METHOD PUBLIC Clone : I_Node
VAR
    pNode : POINTER TO Node_F_VN_ConvertMaps;
END_VAR
pNode := __NEW(Node_F_VN_ConvertMaps);
Clone := pNode^;
END_METHOD

METHOD PROTECTED OnExecute
hresult.Value := F_VN_ConvertMaps(
    ipSrcMap1 := ipSrcMap1.Value,
    ipSrcMap2 := ipSrcMap2.Value,
    ipDestMap1 := ipDestMap1.Value,
    ipDestMap2 := ipDestMap2.Value,
    eDestMap1Type := eDestMap1Type.Value,
    nDestMap1Channels := nDestMap1Channels.Value,
    hrPrev := hrPrev.Value);
END_METHOD

METHOD PUBLIC PreExecutionCheck
VAR_INPUT
    Check : I_PreExecutionChecks;
END_VAR
Check.IsTrue(IsRemapMapPairValid(ipSrcMap1.Value, ipSrcMap2.Value), 'Unsupported source map pair: use REAL XY, separate REAL X/Y, or INT XY with optional UINT coefficients');
Check.IsTrue((eDestMap1Type.Value = ETcVnElementType.TCVN_ET_REAL) OR
             (eDestMap1Type.Value = ETcVnElementType.TCVN_ET_INT), 'Destination map type must be REAL or INT');
Check.IsTrue((nDestMap1Channels.Value = 1) OR (nDestMap1Channels.Value = 2), 'Destination map must have 1 or 2 channels');
Check.IsTrue((eDestMap1Type.Value <> ETcVnElementType.TCVN_ET_INT) OR
             (nDestMap1Channels.Value = 2), 'Fixed-point destination map must have 2 channels');
Check.IsTrue((ipDestMap1.Value = 0) OR ((ipDestMap1.Value <> ipSrcMap1.Value) AND (ipDestMap1.Value <> ipSrcMap2.Value)), 'ipDestMap1 must be different from the source maps');
Check.IsTrue((ipDestMap2.Value = 0) OR ((ipDestMap2.Value <> ipSrcMap1.Value) AND (ipDestMap2.Value <> ipSrcMap2.Value)), 'ipDestMap2 must be different from the source maps');
Check.IsTrue((ipDestMap1.Value = 0) OR (ipDestMap1.Value <> ipDestMap2.Value), 'Destination maps must be different images');
END_METHOD

END_FUNCTION_BLOCK

// Nodes/Geometric and Coord Transform/Node_F_VN_ConvertPolarToCartesianImages
{attribute 'linkalways'}
{attribute 'no_explicit_call' := 'This FB is a CLASS and must be accessed using methods or properties'}
{attribute 'enable_dynamic_creation'}
FUNCTION_BLOCK Node_F_VN_ConvertPolarToCartesianImages EXTENDS VisionNode
VAR
    ipSrcImageMag : _ITcVnImage;
    ipSrcImageAng : _ITcVnImage;
    ipDestImageX : _ITcVnImage;
    ipDestImageY : _ITcVnImage;
    hrPrev : _HRESULT(S_OK);
    hresult : _HRESULT(S_OK);
END_VAR

METHOD FB_init : BOOL
VAR_INPUT
    bInitRetains : BOOL;
    bInCopyCode : BOOL;
END_VAR
AddInput('ipSrcImageMag', ipSrcImageMag);
AddInput('ipSrcImageAng', ipSrcImageAng);
AddOutput('ipDestImageX', ipDestImageX);
AddOutput('ipDestImageY', ipDestImageY);
AddInput('hrPrev', hrPrev);
AddOutput('hresult', hresult);
END_METHOD

METHOD PUBLIC Clone : I_Node
VAR
    pNode : POINTER TO Node_F_VN_ConvertPolarToCartesianImages;
END_VAR
pNode := __NEW(Node_F_VN_ConvertPolarToCartesianImages);
Clone := pNode^;
END_METHOD

METHOD PROTECTED OnExecute
hresult.Value := F_VN_ConvertPolarToCartesianImages(
    ipSrcImageMag := ipSrcImageMag.Value,
    ipSrcImageAng := ipSrcImageAng.Value,
    ipDestImageX := ipDestImageX.Value,
    ipDestImageY := ipDestImageY.Value,
    hrPrev := hrPrev.Value);
END_METHOD

METHOD PUBLIC PreExecutionCheck
VAR_INPUT
    Check : I_PreExecutionChecks;
END_VAR
Check.IsTrue(ipSrcImageMag.IsValid, 'ipSrcImageMag must contain an image');
Check.IsTrue(ipSrcImageMag.IsElementType(ETcVnElementType.TCVN_ET_REAL) OR
             ipSrcImageMag.IsElementType(ETcVnElementType.TCVN_ET_LREAL), 'Coordinate images must contain REAL or LREAL elements');
Check.IsTrue(ipSrcImageAng.IsValid, 'ipSrcImageAng must contain an image');
Check.IsTrue(ImagesHaveMatchingPixelFormats(ipSrcImageMag.Value, ipSrcImageAng.Value), 'Source images must have matching pixel formats');
Check.IsTrue(IsImage1SizeEqualToImage2Size(ipSrcImageMag.Value, ipSrcImageAng.Value), 'Source images must have matching dimensions');
END_METHOD

END_FUNCTION_BLOCK

// Nodes/Geometric and Coord Transform/Node_F_VN_ConvertPolarToCartesianImagesExp
{attribute 'linkalways'}
{attribute 'no_explicit_call' := 'This FB is a CLASS and must be accessed using methods or properties'}
{attribute 'enable_dynamic_creation'}
FUNCTION_BLOCK Node_F_VN_ConvertPolarToCartesianImagesExp EXTENDS VisionNode
VAR
    ipSrcImageMag : _ITcVnImage;
    ipSrcImageAng : _ITcVnImage;
    ipDestImageX : _ITcVnImage;
    ipDestImageY : _ITcVnImage;
    bAngleInDegrees : _BOOL(FALSE);
    hrPrev : _HRESULT(S_OK);
    hresult : _HRESULT(S_OK);
END_VAR

METHOD FB_init : BOOL
VAR_INPUT
    bInitRetains : BOOL;
    bInCopyCode : BOOL;
END_VAR
AddInput('ipSrcImageMag', ipSrcImageMag);
AddInput('ipSrcImageAng', ipSrcImageAng);
AddOutput('ipDestImageX', ipDestImageX);
AddOutput('ipDestImageY', ipDestImageY);
AddParameter('bAngleInDegrees', bAngleInDegrees);
AddInput('hrPrev', hrPrev);
AddOutput('hresult', hresult);
END_METHOD

METHOD PUBLIC Clone : I_Node
VAR
    pNode : POINTER TO Node_F_VN_ConvertPolarToCartesianImagesExp;
END_VAR
pNode := __NEW(Node_F_VN_ConvertPolarToCartesianImagesExp);
Clone := pNode^;
END_METHOD

METHOD PROTECTED OnExecute
hresult.Value := F_VN_ConvertPolarToCartesianImagesExp(
    ipSrcImageMag := ipSrcImageMag.Value,
    ipSrcImageAng := ipSrcImageAng.Value,
    ipDestImageX := ipDestImageX.Value,
    ipDestImageY := ipDestImageY.Value,
    bAngleInDegrees := bAngleInDegrees.Value,
    hrPrev := hrPrev.Value);
END_METHOD

METHOD PUBLIC PreExecutionCheck
VAR_INPUT
    Check : I_PreExecutionChecks;
END_VAR
Check.IsTrue(ipSrcImageMag.IsValid, 'ipSrcImageMag must contain an image');
Check.IsTrue(ipSrcImageMag.IsElementType(ETcVnElementType.TCVN_ET_REAL) OR
             ipSrcImageMag.IsElementType(ETcVnElementType.TCVN_ET_LREAL), 'Coordinate images must contain REAL or LREAL elements');
Check.IsTrue(ipSrcImageAng.IsValid, 'ipSrcImageAng must contain an image');
Check.IsTrue(ImagesHaveMatchingPixelFormats(ipSrcImageMag.Value, ipSrcImageAng.Value), 'Source images must have matching pixel formats');
Check.IsTrue(IsImage1SizeEqualToImage2Size(ipSrcImageMag.Value, ipSrcImageAng.Value), 'Source images must have matching dimensions');
END_METHOD

END_FUNCTION_BLOCK

// Nodes/Geometric and Coord Transform/Node_F_VN_ConvertPolarToCartesianPoints
{attribute 'linkalways'} 
{attribute 'no_explicit_call' := 'This FB is a CLASS and must be accessed using methods or properties'}
{attribute 'enable_dynamic_creation'}
FUNCTION_BLOCK Node_F_VN_ConvertPolarToCartesianPoints EXTENDS VisionNode
VAR
	ipSrcPointsPolar : _ITcVnContainer;
    ipDestPointsCart : _ITcVnContainer;
    hrPrev : _HRESULT(S_OK);
	hresult : _HRESULT(S_OK);
END_VAR

METHOD FB_init : BOOL
VAR_INPUT
	bInitRetains : BOOL; // if TRUE, the retain variables are initialized (warm start / cold start)
	bInCopyCode : BOOL;  // if TRUE, the instance afterwards gets moved into the copy code (online change)
END_VAR
AddInput('ipSrcPointsPolar', ipSrcPointsPolar);
AddInput('hrPrev', hrPrev);
AddOutput('ipDestPointsCart', ipDestPointsCart);
AddOutput('hresult',hresult);
END_METHOD

METHOD PUBLIC  Clone : I_Node
VAR
	pNode : POINTER TO Node_F_VN_ConvertPolarToCartesianPoints;
END_VAR
pNode := __NEW(Node_F_VN_ConvertPolarToCartesianPoints);
Clone := pNode^;
END_METHOD

METHOD PROTECTED OnExecute
hresult.Value := F_VN_ConvertPolarToCartesianPoints(
	ipSrcPointsPolar := ipSrcPointsPolar.Value,
	ipDestPointsCart := ipDestPointsCart.Value,
	hrPrev := hrPrev.Value);
END_METHOD

METHOD PUBLIC PreExecutionCheck
VAR_INPUT
	Check : I_PreExecutionChecks;
END_VAR
Check.IsTrue(ipSrcPointsPolar.IsValid, 'ipSrcPointsPolar must be a valid container');
Check.IsTrue((ipSrcPointsPolar.IsType(TC_GLOBAL_CONST_LIST.ContainerType_Vector_TcVnPoint2_REAL) OR
              ipSrcPointsPolar.IsType(TC_GLOBAL_CONST_LIST.ContainerType_Vector_TcVnPoint2_LREAL)),
              'ipSrcPointsPolar contains incorrect type');
END_METHOD

END_FUNCTION_BLOCK

// Nodes/Geometric and Coord Transform/Node_F_VN_ConvertPolarToCartesianPointsExp
{attribute 'linkalways'} 
{attribute 'no_explicit_call' := 'This FB is a CLASS and must be accessed using methods or properties'}
{attribute 'enable_dynamic_creation'}
FUNCTION_BLOCK Node_F_VN_ConvertPolarToCartesianPointsExp EXTENDS VisionNode
VAR
	ipSrcPointsPolar : _ITcVnContainer;
    ipDestPointsCart : _ITcVnContainer;
    bAngleInDegrees : _BOOL(FALSE);
    hrPrev : _HRESULT(S_OK);
	hresult : _HRESULT(S_OK);
END_VAR

METHOD FB_init : BOOL
VAR_INPUT
	bInitRetains : BOOL; // if TRUE, the retain variables are initialized (warm start / cold start)
	bInCopyCode : BOOL;  // if TRUE, the instance afterwards gets moved into the copy code (online change)
END_VAR
AddInput('ipSrcPointsPolar', ipSrcPointsPolar);
AddParameter('bAngleInDegrees', bAngleInDegrees);
AddInput('hrPrev', hrPrev);
AddOutput('ipDestPointsCart', ipDestPointsCart);
AddOutput('hresult',hresult);
END_METHOD

METHOD PUBLIC  Clone : I_Node
VAR
	pNode : POINTER TO Node_F_VN_ConvertPolarToCartesianPointsExp;
END_VAR
pNode := __NEW(Node_F_VN_ConvertPolarToCartesianPointsExp);
Clone := pNode^;
END_METHOD

METHOD PROTECTED OnExecute
hresult.Value := F_VN_ConvertPolarToCartesianPointsExp(
	ipSrcPointsPolar := ipSrcPointsPolar.Value,
	ipDestPointsCart := ipDestPointsCart.Value,
    bAngleInDegrees := bAngleInDegrees.Value,
	hrPrev := hrPrev.Value);
END_METHOD

METHOD PUBLIC PreExecutionCheck
VAR_INPUT
	Check : I_PreExecutionChecks;
END_VAR
Check.IsTrue(ipSrcPointsPolar.IsValid, 'ipSrcPointsPolar must be a valid container');
Check.IsTrue((ipSrcPointsPolar.IsType(TC_GLOBAL_CONST_LIST.ContainerType_Vector_TcVnPoint2_REAL) OR
              ipSrcPointsPolar.IsType(TC_GLOBAL_CONST_LIST.ContainerType_Vector_TcVnPoint2_LREAL)),
              'ipSrcPointsPolar contains incorrect type');
END_METHOD

END_FUNCTION_BLOCK

// Nodes/Geometric and Coord Transform/Node_F_VN_DecomposeAffineTransformation
{attribute 'linkalways'} 
{attribute 'no_explicit_call' := 'This FB is a CLASS and must be accessed using methods or properties'}
{attribute 'enable_dynamic_creation'}
FUNCTION_BLOCK Node_F_VN_DecomposeAffineTransformation EXTENDS VisionNode
VAR
    aAffineTransform : _TcVnMatrix2x3_LREAL;
    fRotationAngle : _LREAL(0.0);
    hrPrev : _HRESULT(S_OK);
	hresult : _HRESULT(S_OK);
END_VAR

METHOD FB_init : BOOL
VAR_INPUT
	bInitRetains : BOOL; // if TRUE, the retain variables are initialized (warm start / cold start)
	bInCopyCode : BOOL;  // if TRUE, the instance afterwards gets moved into the copy code (online change)
END_VAR
AddInput('aAffineTransform', aAffineTransform);
AddInput('hrPrev', hrPrev);
AddOutput('fRotationAngle', fRotationAngle);
AddOutput('hresult',hresult);
END_METHOD

METHOD PUBLIC  Clone : I_Node
VAR
	pNode : POINTER TO Node_F_VN_DecomposeAffineTransformation;
END_VAR
pNode := __NEW(Node_F_VN_DecomposeAffineTransformation);
Clone := pNode^;
END_METHOD

METHOD PROTECTED OnExecute
hresult.Value := F_VN_DecomposeAffineTransformation(
	aAffineTransform := aAffineTransform.Value, 
	fRotationAngle := fRotationAngle.Value, 
	hrPrev := hrPrev.Value);
END_METHOD

METHOD PUBLIC PreExecutionCheck
VAR_INPUT
	Check : I_PreExecutionChecks;
END_VAR
END_METHOD

END_FUNCTION_BLOCK

// Nodes/Geometric and Coord Transform/Node_F_VN_DecomposeAffineTransformationExp
{attribute 'linkalways'} 
{attribute 'no_explicit_call' := 'This FB is a CLASS and must be accessed using methods or properties'}
{attribute 'enable_dynamic_creation'}
FUNCTION_BLOCK Node_F_VN_DecomposeAffineTransformationExp EXTENDS VisionNode
VAR
    aAffineTransform : _TcVnMatrix2x3_LREAL;
    fRotationAngle : _LREAL(0.0);
    aTranslationVector : _TcVnVector2_LREAL;
    aScaleVector : _TcVnVector2_LREAL;
    aSkewVector : _TcVnVector2_LREAL;
    hrPrev : _HRESULT(S_OK);
	hresult : _HRESULT(S_OK);
END_VAR

METHOD FB_init : BOOL
VAR_INPUT
	bInitRetains : BOOL; // if TRUE, the retain variables are initialized (warm start / cold start)
	bInCopyCode : BOOL;  // if TRUE, the instance afterwards gets moved into the copy code (online change)
END_VAR
AddInput('aAffineTransform', aAffineTransform);
AddInput('hrPrev', hrPrev);
AddOutput('fRotationAngle', fRotationAngle);
AddOutput('aTranslationVector', aTranslationVector);
AddOutput('aScaleVector', aScaleVector);
AddOutput('fRaSkewVectorotationAngle', aSkewVector);
AddOutput('hresult', hresult);
END_METHOD

METHOD PUBLIC  Clone : I_Node
VAR
	pNode : POINTER TO Node_F_VN_DecomposeAffineTransformationExp;
END_VAR
pNode := __NEW(Node_F_VN_DecomposeAffineTransformationExp);
Clone := pNode^;
END_METHOD

METHOD PROTECTED OnExecute
hresult.Value := F_VN_DecomposeAffineTransformationExp(
	aAffineTransform := aAffineTransform.Value,
	fRotationAngle := fRotationAngle.Value,
    aTranslationVector := aTranslationVector.Value,
    aScaleVector := aScaleVector.Value,
    aSkewVector := aSkewVector.Value,
	hrPrev := hrPrev.Value);
END_METHOD

METHOD PUBLIC PreExecutionCheck
VAR_INPUT
	Check : I_PreExecutionChecks;
END_VAR
END_METHOD

END_FUNCTION_BLOCK

// Nodes/Geometric and Coord Transform/Node_F_VN_FlipImage
{attribute 'linkalways'} 
{attribute 'no_explicit_call' := 'This FB is a CLASS and must be accessed using methods or properties'}
{attribute 'enable_dynamic_creation'}
FUNCTION_BLOCK Node_F_VN_FlipImage EXTENDS VisionNode
VAR
	ipSrcImage : _ITcVnImage;
    ipDestImage : _ITcVnImage;
    eFlipAxis : _ETcVnFlipAxis(ETcVnFlipAxis.TCVN_FA_X);
    hrPrev : _HRESULT(S_OK);
	hresult : _HRESULT(S_OK);
END_VAR

METHOD FB_init : BOOL
VAR_INPUT
	bInitRetains : BOOL; // if TRUE, the retain variables are initialized (warm start / cold start)
	bInCopyCode : BOOL;  // if TRUE, the instance afterwards gets moved into the copy code (online change)
END_VAR
AddInput('ipSrcImage', ipSrcImage);
AddInput('hrPrev', hrPrev);
AddOutput('ipDestImage', ipDestImage);
AddOutput('hresult',hresult);
AddParameter('eFlipAxis', eFlipAxis);
END_METHOD

METHOD PUBLIC  Clone : I_Node
VAR
	pNode : POINTER TO Node_F_VN_FlipImage;
END_VAR
pNode := __NEW(Node_F_VN_FlipImage);
Clone := pNode^;
END_METHOD

METHOD PROTECTED OnExecute
hresult.Value := F_VN_FlipImage(
	ipSrcImage := ipSrcImage.Value, 
	ipDestImage := ipDestImage.Value, 
	eFlipAxis := eFlipAxis.Value, 
	hrPrev := hrPrev.Value);
END_METHOD

METHOD PUBLIC PreExecutionCheck
VAR_INPUT
	Check : I_PreExecutionChecks;
END_VAR
Check.IsTrue(ipSrcImage.IsValid, 'ipSrcImage must contain an image');
END_METHOD

END_FUNCTION_BLOCK

// Nodes/Geometric and Coord Transform/Node_F_VN_GenerateAffineTransformationUnitMatrix2D
{attribute 'linkalways'} 
{attribute 'no_explicit_call' := 'This FB is a CLASS and must be accessed using methods or properties'}
{attribute 'enable_dynamic_creation'}
FUNCTION_BLOCK Node_F_VN_GenerateAffineTransformationUnitMatrix2D EXTENDS VisionNode
VAR
    aTransformationMatrix : _TcVnMatrix2x3_LREAL;
    hrPrev : _HRESULT(S_OK);
	hresult : _HRESULT(S_OK);
END_VAR

METHOD FB_init : BOOL
VAR_INPUT
	bInitRetains : BOOL; // if TRUE, the retain variables are initialized (warm start / cold start)
	bInCopyCode : BOOL;  // if TRUE, the instance afterwards gets moved into the copy code (online change)
END_VAR
AddInput('hrPrev', hrPrev);
AddOutput('aTransformationMatrix', aTransformationMatrix);
AddOutput('hresult',hresult);
END_METHOD

METHOD PUBLIC  Clone : I_Node
VAR
	pNode : POINTER TO Node_F_VN_GenerateAffineTransformationUnitMatrix2D;
END_VAR
pNode := __NEW(Node_F_VN_GenerateAffineTransformationUnitMatrix2D);
Clone := pNode^;
END_METHOD

METHOD PROTECTED OnExecute
hresult.Value := F_VN_GenerateAffineTransformationUnitMatrix2D(
	aTransformationMatrix := aTransformationMatrix.Value,
	hrPrev := hrPrev.Value);
END_METHOD

METHOD PUBLIC PreExecutionCheck
VAR_INPUT
	Check : I_PreExecutionChecks;
END_VAR
END_METHOD

END_FUNCTION_BLOCK

// Nodes/Geometric and Coord Transform/Node_F_VN_GetAffineTransformation
{attribute 'linkalways'} 
{attribute 'no_explicit_call' := 'This FB is a CLASS and must be accessed using methods or properties'}
{attribute 'enable_dynamic_creation'}
FUNCTION_BLOCK Node_F_VN_GetAffineTransformation EXTENDS VisionNode
VAR
	aSrcPoints : _TcVnArray3_Point2_REAL;
    aDestPoints : _TcVnArray3_Point2_REAL;
    aTransformationMatrix : _TcVnMatrix2x3_LREAL;
    hrPrev : _HRESULT(S_OK);
	hresult : _HRESULT(S_OK);
END_VAR

METHOD FB_init : BOOL
VAR_INPUT
	bInitRetains : BOOL; // if TRUE, the retain variables are initialized (warm start / cold start)
	bInCopyCode : BOOL;  // if TRUE, the instance afterwards gets moved into the copy code (online change)
END_VAR
AddInput('aSrcPoints', aSrcPoints);
AddInput('aDestPoints', aDestPoints);
AddInput('hrPrev', hrPrev);
AddOutput('aTransformationMatrix', aTransformationMatrix);
AddOutput('hresult',hresult);
END_METHOD

METHOD PUBLIC  Clone : I_Node
VAR
	pNode : POINTER TO Node_F_VN_GetAffineTransformation;
END_VAR
pNode := __NEW(Node_F_VN_GetAffineTransformation);
Clone := pNode^;
END_METHOD

METHOD PROTECTED OnExecute
hresult.Value := F_VN_GetAffineTransformation(
	aSrcPoints := aSrcPoints.Value, 
	aDestPoints := aDestPoints.Value, 
	aTransformationMatrix := aTransformationMatrix.Value, 
	hrPrev := hrPrev.Value);
END_METHOD

METHOD PUBLIC PreExecutionCheck
VAR_INPUT
	Check : I_PreExecutionChecks;
END_VAR
END_METHOD

END_FUNCTION_BLOCK

// Nodes/Geometric and Coord Transform/Node_F_VN_GetAffineTransformation2D
{attribute 'linkalways'} 
{attribute 'no_explicit_call' := 'This FB is a CLASS and must be accessed using methods or properties'}
{attribute 'enable_dynamic_creation'}
FUNCTION_BLOCK Node_F_VN_GetAffineTransformation2D EXTENDS VisionNode
VAR
	ipSrcPoints : _ITcVnContainer;
    ipDestPoints : _ITcVnContainer;
    aAffineTransform : _TcVnMatrix2x3_LREAL;
    hrPrev : _HRESULT(S_OK);
	hresult : _HRESULT(S_OK);
END_VAR

METHOD FB_init : BOOL
VAR_INPUT
	bInitRetains : BOOL; // if TRUE, the retain variables are initialized (warm start / cold start)
	bInCopyCode : BOOL;  // if TRUE, the instance afterwards gets moved into the copy code (online change)
END_VAR
AddInput('ipSrcPoints', ipSrcPoints);
AddInput('ipDestPoints', ipDestPoints);
AddInput('hrPrev', hrPrev);
AddOutput('aAffineTransform', aAffineTransform);
AddOutput('hresult',hresult);
END_METHOD

METHOD PUBLIC  Clone : I_Node
VAR
	pNode : POINTER TO Node_F_VN_GetAffineTransformation2D
;
END_VAR
pNode := __NEW(Node_F_VN_GetAffineTransformation2D);
Clone := pNode^;
END_METHOD

METHOD PROTECTED OnExecute
hresult.Value := F_VN_GetAffineTransformation2D(
	ipSrcPoints := ipSrcPoints.Value,
	ipDestPoints := ipDestPoints.Value,
	aAffineTransform := aAffineTransform.Value,
	hrPrev := hrPrev.Value);
END_METHOD

METHOD PUBLIC PreExecutionCheck
VAR_INPUT
	Check : I_PreExecutionChecks;
END_VAR
VAR
    elementNum : ULINT;
END_VAR
Check.IsTrue(ipSrcPoints.IsValid, 'ipSrcPoints must be a valid container');
Check.IsTrue(ipSrcPoints.IsType(TC_GLOBAL_CONST_LIST.ContainerType_Vector_TcVnPoint2_REAL), 'ipSrcPoints contains incorrect type');
Check.IsTrue((ipSrcPoints.TryGetElementNum(elementNum) AND (elementNum >= 3)), 'ipSrcPoints must contain at least 3 points');
END_METHOD

END_FUNCTION_BLOCK

// Nodes/Geometric and Coord Transform/Node_F_VN_GetPerspectiveTransformation
{attribute 'linkalways'} 
{attribute 'no_explicit_call' := 'This FB is a CLASS and must be accessed using methods or properties'}
{attribute 'enable_dynamic_creation'}
FUNCTION_BLOCK Node_F_VN_GetPerspectiveTransformation EXTENDS VisionNode
VAR
	aSrcPoints : _TcVnArray4_Point2_REAL;
    aDestPoints : _TcVnArray4_Point2_REAL;
    aTransformationMatrix : _TcVnMatrix3x3_LREAL;
    hrPrev : _HRESULT(S_OK);
	hresult : _HRESULT(S_OK);
END_VAR

METHOD FB_init : BOOL
VAR_INPUT
	bInitRetains : BOOL; // if TRUE, the retain variables are initialized (warm start / cold start)
	bInCopyCode : BOOL;  // if TRUE, the instance afterwards gets moved into the copy code (online change)
END_VAR
AddInput('aSrcPoints', aSrcPoints);
AddInput('aDestPoints', aDestPoints);
AddInput('hrPrev', hrPrev);
AddOutput('aTransformationMatrix', aTransformationMatrix);
AddOutput('hresult',hresult);
END_METHOD

METHOD PUBLIC  Clone : I_Node
VAR
	pNode : POINTER TO Node_F_VN_GetPerspectiveTransformation;
END_VAR
pNode := __NEW(Node_F_VN_GetPerspectiveTransformation);
Clone := pNode^;
END_METHOD

METHOD PROTECTED OnExecute
hresult.Value := F_VN_GetPerspectiveTransformation(
	aSrcPoints := aSrcPoints.Value, 
	aDestPoints := aDestPoints.Value, 
	aTransformationMatrix := aTransformationMatrix.Value, 
	hrPrev := hrPrev.Value);
END_METHOD

METHOD PUBLIC PreExecutionCheck
VAR_INPUT
	Check : I_PreExecutionChecks;
END_VAR
END_METHOD

END_FUNCTION_BLOCK

// Nodes/Geometric and Coord Transform/Node_F_VN_Homography
{attribute 'linkalways'} 
{attribute 'no_explicit_call' := 'This FB is a CLASS and must be accessed using methods or properties'}
{attribute 'enable_dynamic_creation'}
FUNCTION_BLOCK Node_F_VN_Homography EXTENDS VisionNode
VAR
	ipSrcPoints : _ITcVnContainer;
    ipDestPoints : _ITcVnContainer;
    aPerspectiveTransform : _TcVnMatrix3x3_LREAL;
    hrPrev : _HRESULT(S_OK);
	hresult : _HRESULT(S_OK);
END_VAR

METHOD FB_init : BOOL
VAR_INPUT
	bInitRetains : BOOL; // if TRUE, the retain variables are initialized (warm start / cold start)
	bInCopyCode : BOOL;  // if TRUE, the instance afterwards gets moved into the copy code (online change)
END_VAR
AddInput('ipSrcPoints', ipSrcPoints);
AddInput('ipDestPoints', ipDestPoints);
AddInput('hrPrev', hrPrev);
AddOutput('aPerspectiveTransform', aPerspectiveTransform);
AddOutput('hresult', hresult);
END_METHOD

METHOD PUBLIC  Clone : I_Node
VAR
	pNode : POINTER TO Node_F_VN_Homography;
END_VAR
pNode := __NEW(Node_F_VN_Homography);
Clone := pNode^;
END_METHOD

METHOD PROTECTED OnExecute
hresult.Value := F_VN_Homography(
	ipSrcPoints := ipSrcPoints.Value, 
	ipDestPoints := ipDestPoints.Value, 
	aPerspectiveTransform := aPerspectiveTransform.Value, 
	hrPrev := hrPrev.Value);
END_METHOD

METHOD PUBLIC PreExecutionCheck
VAR_INPUT
	Check : I_PreExecutionChecks;
END_VAR
VAR
    elementNumSrc : ULINT;
    elementNumDest : ULINT;
END_VAR
Check.IsTrue(ipSrcPoints.IsValid, 'ipSrcPoints must be a valid container');
Check.IsTrue(ipSrcPoints.IsType(TC_GLOBAL_CONST_LIST.ContainerType_Vector_TcVnPoint2_REAL), 'ipSrcPoints contains incorrect type');

ipSrcPoints.TryGetElementNum(elementNumSrc);
Check.IsTrue(elementNumSrc >= 4, 'ipSrcPoints must contain at least 4 elements');

Check.IsTrue(ipDestPoints.IsValid, 'ipDestPoints must be a valid container');
Check.IsTrue(ipDestPoints.IsType(TC_GLOBAL_CONST_LIST.ContainerType_Vector_TcVnPoint2_REAL), 'ipDestPoints contains incorrect type');

ipDestPoints.TryGetElementNum(elementNumDest);
Check.IsTrue(elementNumSrc = elementNumDest, 'ipDestPoints must contain the same number of elements as ipSrcPoints');
END_METHOD

END_FUNCTION_BLOCK

// Nodes/Geometric and Coord Transform/Node_F_VN_HomographyExp
{attribute 'linkalways'} 
{attribute 'no_explicit_call' := 'This FB is a CLASS and must be accessed using methods or properties'}
{attribute 'enable_dynamic_creation'}
FUNCTION_BLOCK Node_F_VN_HomographyExp EXTENDS VisionNode
VAR
	ipSrcPoints : _ITcVnContainer;
    ipDestPoints : _ITcVnContainer;
    aPerspectiveTransform : _TcVnMatrix3x3_LREAL;
    eAlgorithm : _ETcVnEstimationAlgorithm(ETcVnEstimationAlgorithm.TCVN_EA_DEFAULT);
    fReprojThreshold : _LREAL(0.0);
    ipInlierMask : _ITcVnContainer;
    nMaxIterations : _UDINT(0);
    fConfidence : _LREAL(0.0);
    hrPrev : _HRESULT(S_OK);
	hresult : _HRESULT(S_OK);
END_VAR

METHOD FB_init : BOOL
VAR_INPUT
	bInitRetains : BOOL; // if TRUE, the retain variables are initialized (warm start / cold start)
	bInCopyCode : BOOL;  // if TRUE, the instance afterwards gets moved into the copy code (online change)
END_VAR
AddInput('ipSrcPoints', ipSrcPoints);
AddInput('ipDestPoints', ipDestPoints);
AddParameter('eAlgorithm', eAlgorithm);
AddParameter('fReprojThreshold', fReprojThreshold);
AddParameter('nMaxIterations', nMaxIterations);
AddParameter('fConfidence', fConfidence);
AddInput('hrPrev', hrPrev);
AddOutput('aPerspectiveTransform', aPerspectiveTransform);
AddOutput('ipInlierMask', ipInlierMask);
AddOutput('hresult', hresult);
END_METHOD

METHOD PUBLIC  Clone : I_Node
VAR
	pNode : POINTER TO Node_F_VN_HomographyExp;
END_VAR
pNode := __NEW(Node_F_VN_HomographyExp);
Clone := pNode^;
END_METHOD

METHOD PROTECTED OnExecute
hresult.Value := F_VN_HomographyExp(
	ipSrcPoints := ipSrcPoints.Value,
	ipDestPoints := ipDestPoints.Value,
	aPerspectiveTransform := aPerspectiveTransform.Value,
    eAlgorithm := eAlgorithm.Value,
    fReprojThreshold := fReprojThreshold.Value,
    ipInlierMask := ipInlierMask.Value,
    nMaxIterations := nMaxIterations.Value,
    fConfidence := fConfidence.Value,
	hrPrev := hrPrev.Value);
END_METHOD

METHOD PUBLIC PreExecutionCheck
VAR_INPUT
	Check : I_PreExecutionChecks;
END_VAR
VAR
    elementNumSrc : ULINT;
    elementNumDest : ULINT;
END_VAR
Check.IsTrue(ipSrcPoints.IsValid, 'ipSrcPoints must be a valid container');
Check.IsTrue(ipSrcPoints.IsType(TC_GLOBAL_CONST_LIST.ContainerType_Vector_TcVnPoint2_REAL), 'ipSrcPoints contains incorrect type');

ipSrcPoints.TryGetElementNum(elementNumSrc);
Check.IsTrue(elementNumSrc >= 4, 'ipSrcPoints must contain at least 4 elements');

Check.IsTrue(ipDestPoints.IsValid, 'ipDestPoints must be a valid container');
Check.IsTrue(ipDestPoints.IsType(TC_GLOBAL_CONST_LIST.ContainerType_Vector_TcVnPoint2_REAL), 'ipDestPoints contains incorrect type');

ipDestPoints.TryGetElementNum(elementNumDest);
Check.IsTrue(elementNumSrc = elementNumDest, 'ipDestPoints must contain the same number of elements as ipSrcPoints');

Check.IsFalse((fConfidence.Value >= 0 OR fConfidence.Value <= 1), 'fConfidence must be between 0 and 1');
END_METHOD

END_FUNCTION_BLOCK

// Nodes/Geometric and Coord Transform/Node_F_VN_InvertAffineTransformation
{attribute 'linkalways'} 
{attribute 'no_explicit_call' := 'This FB is a CLASS and must be accessed using methods or properties'}
{attribute 'enable_dynamic_creation'}
FUNCTION_BLOCK Node_F_VN_InvertAffineTransformation EXTENDS VisionNode
VAR
    aTransformationMatrix : _TcVnMatrix2x3_LREAL;
    aInvertedTransformationMatrix : _TcVnMatrix2x3_LREAL;
    hrPrev : _HRESULT(S_OK);
	hresult : _HRESULT(S_OK);
END_VAR

METHOD FB_init : BOOL
VAR_INPUT
	bInitRetains : BOOL; // if TRUE, the retain variables are initialized (warm start / cold start)
	bInCopyCode : BOOL;  // if TRUE, the instance afterwards gets moved into the copy code (online change)
END_VAR
AddInput('aTransformationMatrix', aTransformationMatrix);
AddInput('hrPrev', hrPrev);
AddOutput('aInvertedTransformationMatrix', aInvertedTransformationMatrix);
AddOutput('hresult',hresult);
END_METHOD

METHOD PUBLIC  Clone : I_Node
VAR
	pNode : POINTER TO Node_F_VN_InvertAffineTransformation;
END_VAR
pNode := __NEW(Node_F_VN_InvertAffineTransformation);
Clone := pNode^;
END_METHOD

METHOD PROTECTED OnExecute
hresult.Value := F_VN_InvertAffineTransformation(
	aTransformationMatrix := aTransformationMatrix.Value,
    aInvertedTransformationMatrix := aInvertedTransformationMatrix.Value,
	hrPrev := hrPrev.Value);
END_METHOD

METHOD PUBLIC PreExecutionCheck
VAR_INPUT
	Check : I_PreExecutionChecks;
END_VAR
END_METHOD

END_FUNCTION_BLOCK

// Nodes/Geometric and Coord Transform/Node_F_VN_PerspectiveTransformation
{attribute 'linkalways'} 
{attribute 'no_explicit_call' := 'This FB is a CLASS and must be accessed using methods or properties'}
{attribute 'enable_dynamic_creation'}
FUNCTION_BLOCK Node_F_VN_PerspectiveTransformation EXTENDS VisionNode
VAR
	ipSrcPoints : _ITcVnContainer;
    ipDestPoints : _ITcVnContainer;
    aRotationMatrix : _TcVnMatrix3x3_LREAL;
    aTranslationVector : _TcVnVector3_LREAL;
    hrPrev : _HRESULT(S_OK);
	hresult : _HRESULT(S_OK);
END_VAR

METHOD FB_init : BOOL
VAR_INPUT
	bInitRetains : BOOL; // if TRUE, the retain variables are initialized (warm start / cold start)
	bInCopyCode : BOOL;  // if TRUE, the instance afterwards gets moved into the copy code (online change)
END_VAR
AddInput('ipSrcPoints', ipSrcPoints);
AddInput('aRotationMatrix', aRotationMatrix);
AddInput('aTranslationVector', aTranslationVector);
AddInput('hrPrev', hrPrev);
AddOutput('ipDestPoints', ipDestPoints);
AddOutput('hresult',hresult);
END_METHOD

METHOD PUBLIC  Clone : I_Node
VAR
	pNode : POINTER TO Node_F_VN_PerspectiveTransformation;
END_VAR
pNode := __NEW(Node_F_VN_PerspectiveTransformation);
Clone := pNode^;
END_METHOD

METHOD PROTECTED OnExecute
hresult.Value := F_VN_PerspectiveTransformation(
	ipSrcPoints := ipSrcPoints.Value,
	ipDestPoints := ipDestPoints.Value,
	aRotationMatrix := aRotationMatrix.Value,
    aTranslationVector := aTranslationVector.Value,
	hrPrev := hrPrev.Value);
END_METHOD

METHOD PUBLIC PreExecutionCheck
VAR_INPUT
	Check : I_PreExecutionChecks;
END_VAR
Check.IsTrue(ipSrcPoints.IsValid, 'ipSrcPoints must be a valid container');
Check.IsTrue((ipSrcPoints.IsType(TC_GLOBAL_CONST_LIST.ContainerType_Vector_TcVnPoint3_REAL) OR
              ipSrcPoints.IsType(TC_GLOBAL_CONST_LIST.ContainerType_Vector_TcVnPoint3_LREAL)),
              'ipSrcPoints contains incorrect type');
END_METHOD

END_FUNCTION_BLOCK

// Nodes/Geometric and Coord Transform/Node_F_VN_PyramidDown
{attribute 'linkalways'} 
{attribute 'no_explicit_call' := 'This FB is a CLASS and must be accessed using methods or properties'}
{attribute 'enable_dynamic_creation'}
FUNCTION_BLOCK Node_F_VN_PyramidDown EXTENDS VisionNode
VAR
    ipSrcImage : _ITcVnImage;
    ipDestImage : _ITcVnImage;
    hrPrev : _HRESULT(S_OK);
	hresult : _HRESULT(S_OK);
END_VAR

METHOD FB_init : BOOL
VAR_INPUT
	bInitRetains : BOOL; // if TRUE, the retain variables are initialized (warm start / cold start)
	bInCopyCode : BOOL;  // if TRUE, the instance afterwards gets moved into the copy code (online change)
END_VAR
AddInput('ipSrcImage', ipSrcImage);
AddInput('hrPrev', hrPrev);
AddOutput('ipDestImage', ipDestImage);
AddOutput('hresult',hresult);
END_METHOD

METHOD PUBLIC  Clone : I_Node
VAR
	pNode : POINTER TO Node_F_VN_PyramidDown;
END_VAR
pNode := __NEW(Node_F_VN_PyramidDown);
Clone := pNode^;
END_METHOD

METHOD PROTECTED OnExecute
hresult.Value := F_VN_PyramidDown(
    ipSrcImage := ipSrcImage.Value,
	ipDestImage := ipDestImage.Value,
	hrPrev:= hrPrev.Value);
END_METHOD

METHOD PUBLIC PreExecutionCheck
VAR_INPUT
	Check : I_PreExecutionChecks;
END_VAR
Check.IsTrue(ipSrcImage.IsValid, 'ipSrcImage must contain an image');
END_METHOD

END_FUNCTION_BLOCK

// Nodes/Geometric and Coord Transform/Node_F_VN_PyramidUp
{attribute 'linkalways'} 
{attribute 'no_explicit_call' := 'This FB is a CLASS and must be accessed using methods or properties'}
{attribute 'enable_dynamic_creation'}
FUNCTION_BLOCK Node_F_VN_PyramidUp EXTENDS VisionNode
VAR
    ipSrcImage : _ITcVnImage;
    ipDestImage : _ITcVnImage;
    hrPrev : _HRESULT(S_OK);
	hresult : _HRESULT(S_OK);
END_VAR

METHOD FB_init : BOOL
VAR_INPUT
	bInitRetains : BOOL; // if TRUE, the retain variables are initialized (warm start / cold start)
	bInCopyCode : BOOL;  // if TRUE, the instance afterwards gets moved into the copy code (online change)
END_VAR
AddInput('ipSrcImage', ipSrcImage);
AddInput('hrPrev', hrPrev);
AddOutput('ipDestImage', ipDestImage);
AddOutput('hresult',hresult);
END_METHOD

METHOD PUBLIC  Clone : I_Node
VAR
	pNode : POINTER TO Node_F_VN_PyramidUp;
END_VAR
pNode := __NEW(Node_F_VN_PyramidUp);
Clone := pNode^;
END_METHOD

METHOD PROTECTED OnExecute
hresult.Value := F_VN_PyramidUp(
    ipSrcImage := ipSrcImage.Value,
	ipDestImage := ipDestImage.Value,
	hrPrev:= hrPrev.Value);
END_METHOD

METHOD PUBLIC PreExecutionCheck
VAR_INPUT
	Check : I_PreExecutionChecks;
END_VAR
Check.IsTrue(ipSrcImage.IsValid, 'ipSrcImage must contain an image');
END_METHOD

END_FUNCTION_BLOCK

// Nodes/Geometric and Coord Transform/Node_F_VN_RemapImage
{attribute 'linkalways'}
{attribute 'no_explicit_call' := 'This FB is a CLASS and must be accessed using methods or properties'}
{attribute 'enable_dynamic_creation'}
FUNCTION_BLOCK Node_F_VN_RemapImage EXTENDS VisionNode
VAR
    ipSrcImage : _ITcVnImage;
    ipDestImage : _ITcVnImage;
    ipMap1 : _ITcVnImage;
    ipMap2 : _ITcVnImage;
    hrPrev : _HRESULT(S_OK);
    hresult : _HRESULT(S_OK);
END_VAR

METHOD FB_init : BOOL
VAR_INPUT
    bInitRetains : BOOL;
    bInCopyCode : BOOL;
END_VAR
AddInput('ipSrcImage', ipSrcImage);
AddOutput('ipDestImage', ipDestImage);
AddInput('ipMap1', ipMap1);
AddInput('ipMap2', ipMap2);
AddInput('hrPrev', hrPrev);
AddOutput('hresult', hresult);
END_METHOD

METHOD PUBLIC Clone : I_Node
VAR
    pNode : POINTER TO Node_F_VN_RemapImage;
END_VAR
pNode := __NEW(Node_F_VN_RemapImage);
Clone := pNode^;
END_METHOD

METHOD PROTECTED OnExecute
hresult.Value := F_VN_RemapImage(
    ipSrcImage := ipSrcImage.Value,
    ipDestImage := ipDestImage.Value,
    ipMap1 := ipMap1.Value,
    ipMap2 := ipMap2.Value,
    hrPrev := hrPrev.Value);
END_METHOD

METHOD PUBLIC PreExecutionCheck
VAR_INPUT
    Check : I_PreExecutionChecks;
END_VAR
Check.IsTrue(ipSrcImage.IsValid, 'ipSrcImage must contain an image');
Check.IsTrue((ipDestImage.Value = 0) OR (ipDestImage.Value <> ipSrcImage.Value), 'Destination must be different from the source image');
Check.IsTrue(IsRemapMapPairValid(ipMap1.Value, ipMap2.Value), 'Unsupported remap pair: use REAL XY, separate REAL X/Y, or INT XY with optional UINT coefficients');
END_METHOD

END_FUNCTION_BLOCK

// Nodes/Geometric and Coord Transform/Node_F_VN_RemapImageExp
{attribute 'linkalways'}
{attribute 'no_explicit_call' := 'This FB is a CLASS and must be accessed using methods or properties'}
{attribute 'enable_dynamic_creation'}
FUNCTION_BLOCK Node_F_VN_RemapImageExp EXTENDS VisionNode
VAR
    ipSrcImage : _ITcVnImage;
    ipDestImage : _ITcVnImage;
    ipMap1 : _ITcVnImage;
    ipMap2 : _ITcVnImage;
    bRelativeMap : _BOOL(FALSE);
    eInterpolationType : _ETcVnInterpolationType(ETcVnInterpolationType.TCVN_IT_BILINEAR);
    eBorderInterpolation : _ETcVnBorderInterpolationMethod(ETcVnBorderInterpolationMethod.TCVN_BIM_CONSTANT);
    aBorderValue : _TcVnVector4_LREAL;
    hrPrev : _HRESULT(S_OK);
    hresult : _HRESULT(S_OK);
END_VAR

METHOD FB_init : BOOL
VAR_INPUT
    bInitRetains : BOOL;
    bInCopyCode : BOOL;
END_VAR
AddInput('ipSrcImage', ipSrcImage);
AddOutput('ipDestImage', ipDestImage);
AddInput('ipMap1', ipMap1);
AddInput('ipMap2', ipMap2);
AddParameter('bRelativeMap', bRelativeMap);
AddParameter('eInterpolationType', eInterpolationType);
AddParameter('eBorderInterpolation', eBorderInterpolation);
AddInput('aBorderValue', aBorderValue);
AddInput('hrPrev', hrPrev);
AddOutput('hresult', hresult);
END_METHOD

METHOD PUBLIC Clone : I_Node
VAR
    pNode : POINTER TO Node_F_VN_RemapImageExp;
END_VAR
pNode := __NEW(Node_F_VN_RemapImageExp);
Clone := pNode^;
END_METHOD

METHOD PROTECTED OnExecute
hresult.Value := F_VN_RemapImageExp(
    ipSrcImage := ipSrcImage.Value,
    ipDestImage := ipDestImage.Value,
    ipMap1 := ipMap1.Value,
    ipMap2 := ipMap2.Value,
    bRelativeMap := bRelativeMap.Value,
    eInterpolationType := eInterpolationType.Value,
    eBorderInterpolation := eBorderInterpolation.Value,
    aBorderValue := aBorderValue.Value,
    hrPrev := hrPrev.Value);
END_METHOD

METHOD PUBLIC PreExecutionCheck
VAR_INPUT
    Check : I_PreExecutionChecks;
END_VAR
Check.IsTrue(ipSrcImage.IsValid, 'ipSrcImage must contain an image');
Check.IsTrue((ipDestImage.Value = 0) OR (ipDestImage.Value <> ipSrcImage.Value), 'Destination must be different from the source image');
Check.IsTrue(IsRemapMapPairValid(ipMap1.Value, ipMap2.Value), 'Unsupported remap pair: use REAL XY, separate REAL X/Y, or INT XY with optional UINT coefficients');
Check.IsTrue((eInterpolationType.Value = ETcVnInterpolationType.TCVN_IT_NEAREST_NEIGHBOR) OR
             (eInterpolationType.Value = ETcVnInterpolationType.TCVN_IT_BILINEAR) OR
             (eInterpolationType.Value = ETcVnInterpolationType.TCVN_IT_BICUBIC) OR
             (eInterpolationType.Value = ETcVnInterpolationType.TCVN_IT_LANCZOS4), 'Unsupported eInterpolationType');
Check.IsTrue((eBorderInterpolation.Value = ETcVnBorderInterpolationMethod.TCVN_BIM_CONSTANT) OR
             (eBorderInterpolation.Value = ETcVnBorderInterpolationMethod.TCVN_BIM_REPLICATE) OR
             (eBorderInterpolation.Value = ETcVnBorderInterpolationMethod.TCVN_BIM_REFLECT) OR
             (eBorderInterpolation.Value = ETcVnBorderInterpolationMethod.TCVN_BIM_WRAP) OR
             (eBorderInterpolation.Value = ETcVnBorderInterpolationMethod.TCVN_BIM_REFLECT_101) OR
             (eBorderInterpolation.Value = ETcVnBorderInterpolationMethod.TCVN_BIM_DEFAULT) OR
             (eBorderInterpolation.Value = ETcVnBorderInterpolationMethod.TCVN_BIM_TRANSPARENT), 'Unsupported eBorderInterpolation');
END_METHOD

END_FUNCTION_BLOCK

// Nodes/Geometric and Coord Transform/Node_F_VN_RemapImageToLogPolarSpace
{attribute 'linkalways'} 
{attribute 'no_explicit_call' := 'This FB is a CLASS and must be accessed using methods or properties'}
{attribute 'enable_dynamic_creation'}
FUNCTION_BLOCK Node_F_VN_RemapImageToLogPolarSpace EXTENDS VisionNode
VAR
    ipSrcImage : _ITcVnImage;
    ipDestImage : _ITcVnImage;
    aCenter : _TcVnPoint2_REAL;
    hrPrev : _HRESULT(S_OK);
	hresult : _HRESULT(S_OK);
END_VAR

METHOD FB_init : BOOL
VAR_INPUT
	bInitRetains : BOOL; // if TRUE, the retain variables are initialized (warm start / cold start)
	bInCopyCode : BOOL;  // if TRUE, the instance afterwards gets moved into the copy code (online change)
END_VAR
AddInput('ipSrcImage', ipSrcImage);
AddInput('aCenter', aCenter);
AddInput('hrPrev', hrPrev);
AddOutput('ipDestImage', ipDestImage);
AddOutput('hresult',hresult);
END_METHOD

METHOD PUBLIC  Clone : I_Node
VAR
	pNode : POINTER TO Node_F_VN_RemapImageToLogPolarSpace;
END_VAR
pNode := __NEW(Node_F_VN_RemapImageToLogPolarSpace);
Clone := pNode^;
END_METHOD

METHOD PROTECTED OnExecute
hresult.Value := F_VN_RemapImageToLogPolarSpace(
    ipSrcImage := ipSrcImage.Value,
	ipDestImage := ipDestImage.Value,
    aCenter := aCenter.Value,
	hrPrev:= hrPrev.Value);
END_METHOD

METHOD PUBLIC PreExecutionCheck
VAR_INPUT
	Check : I_PreExecutionChecks;
END_VAR
Check.IsTrue(ipSrcImage.IsValid, 'ipSrcImage must contain an image');
END_METHOD

END_FUNCTION_BLOCK

// Nodes/Geometric and Coord Transform/Node_F_VN_RemapImageToLogPolarSpaceExp
{attribute 'linkalways'}
{attribute 'no_explicit_call' := 'This FB is a CLASS and must be accessed using methods or properties'}
{attribute 'enable_dynamic_creation'}
FUNCTION_BLOCK Node_F_VN_RemapImageToLogPolarSpaceExp EXTENDS VisionNode
VAR
    ipSrcImage : _ITcVnImage;
    ipDestImage : _ITcVnImage;
    aCenter : _TcVnPoint2_REAL;
    fScale : _LREAL(0);
    eInterpolationType : _ETcVnInterpolationType(ETcVnInterpolationType.TCVN_IT_BILINEAR);
    hrPrev : _HRESULT(S_OK);
    hresult : _HRESULT(S_OK);
END_VAR

METHOD FB_init : BOOL
VAR_INPUT
    bInitRetains : BOOL;
    bInCopyCode : BOOL;
END_VAR
AddInput('ipSrcImage', ipSrcImage);
AddOutput('ipDestImage', ipDestImage);
AddInput('aCenter', aCenter);
AddParameter('fScale', fScale);
AddParameter('eInterpolationType', eInterpolationType);
AddInput('hrPrev', hrPrev);
AddOutput('hresult', hresult);
END_METHOD

METHOD PUBLIC Clone : I_Node
VAR
    pNode : POINTER TO Node_F_VN_RemapImageToLogPolarSpaceExp;
END_VAR
pNode := __NEW(Node_F_VN_RemapImageToLogPolarSpaceExp);
Clone := pNode^;
END_METHOD

METHOD PROTECTED OnExecute
hresult.Value := F_VN_RemapImageToLogPolarSpaceExp(
    ipSrcImage := ipSrcImage.Value,
    ipDestImage := ipDestImage.Value,
    aCenter := aCenter.Value,
    fScale := fScale.Value,
    eInterpolationType := eInterpolationType.Value,
    hrPrev := hrPrev.Value);
END_METHOD

METHOD PUBLIC PreExecutionCheck
VAR_INPUT
    Check : I_PreExecutionChecks;
END_VAR
Check.IsTrue(ipSrcImage.IsValid, 'ipSrcImage must contain an image');
Check.IsTrue((ipDestImage.Value = 0) OR (ipDestImage.Value <> ipSrcImage.Value), 'Destination must be different from the source image');
Check.IsTrue((eInterpolationType.Value = ETcVnInterpolationType.TCVN_IT_NEAREST_NEIGHBOR) OR
             (eInterpolationType.Value = ETcVnInterpolationType.TCVN_IT_BILINEAR) OR
             (eInterpolationType.Value = ETcVnInterpolationType.TCVN_IT_BICUBIC) OR
             (eInterpolationType.Value = ETcVnInterpolationType.TCVN_IT_AREA_BASED) OR
             (eInterpolationType.Value = ETcVnInterpolationType.TCVN_IT_LANCZOS4), 'Unsupported eInterpolationType');
END_METHOD

END_FUNCTION_BLOCK

// Nodes/Geometric and Coord Transform/Node_F_VN_RemapImageToLogPolarSpaceExp2
{attribute 'linkalways'}
{attribute 'no_explicit_call' := 'This FB is a CLASS and must be accessed using methods or properties'}
{attribute 'enable_dynamic_creation'}
FUNCTION_BLOCK Node_F_VN_RemapImageToLogPolarSpaceExp2 EXTENDS VisionNode
VAR
    ipSrcImage : _ITcVnImage;
    ipDestImage : _ITcVnImage;
    aCenter : _TcVnPoint2_REAL;
    fScale : _LREAL(0);
    eInterpolationType : _ETcVnInterpolationType(ETcVnInterpolationType.TCVN_IT_BILINEAR);
    nDestWidth : _DINT(-1);
    nDestHeight : _DINT(-1);
    hrPrev : _HRESULT(S_OK);
    hresult : _HRESULT(S_OK);
END_VAR

METHOD FB_init : BOOL
VAR_INPUT
    bInitRetains : BOOL;
    bInCopyCode : BOOL;
END_VAR
AddInput('ipSrcImage', ipSrcImage);
AddOutput('ipDestImage', ipDestImage);
AddInput('aCenter', aCenter);
AddParameter('fScale', fScale);
AddParameter('eInterpolationType', eInterpolationType);
AddParameter('nDestWidth', nDestWidth);
AddParameter('nDestHeight', nDestHeight);
AddInput('hrPrev', hrPrev);
AddOutput('hresult', hresult);
END_METHOD

METHOD PUBLIC Clone : I_Node
VAR
    pNode : POINTER TO Node_F_VN_RemapImageToLogPolarSpaceExp2;
END_VAR
pNode := __NEW(Node_F_VN_RemapImageToLogPolarSpaceExp2);
Clone := pNode^;
END_METHOD

METHOD PROTECTED OnExecute
hresult.Value := F_VN_RemapImageToLogPolarSpaceExp2(
    ipSrcImage := ipSrcImage.Value,
    ipDestImage := ipDestImage.Value,
    aCenter := aCenter.Value,
    fScale := fScale.Value,
    eInterpolationType := eInterpolationType.Value,
    nDestWidth := nDestWidth.Value,
    nDestHeight := nDestHeight.Value,
    hrPrev := hrPrev.Value);
END_METHOD

METHOD PUBLIC PreExecutionCheck
VAR_INPUT
    Check : I_PreExecutionChecks;
END_VAR
Check.IsTrue(ipSrcImage.IsValid, 'ipSrcImage must contain an image');
Check.IsTrue((ipDestImage.Value = 0) OR (ipDestImage.Value <> ipSrcImage.Value), 'Destination must be different from the source image');
Check.IsTrue((eInterpolationType.Value = ETcVnInterpolationType.TCVN_IT_NEAREST_NEIGHBOR) OR
             (eInterpolationType.Value = ETcVnInterpolationType.TCVN_IT_BILINEAR) OR
             (eInterpolationType.Value = ETcVnInterpolationType.TCVN_IT_BICUBIC) OR
             (eInterpolationType.Value = ETcVnInterpolationType.TCVN_IT_AREA_BASED) OR
             (eInterpolationType.Value = ETcVnInterpolationType.TCVN_IT_LANCZOS4), 'Unsupported eInterpolationType');
Check.IsTrue(nDestWidth.Value >= -1, 'Destination width must be -1 for source width, 0 for automatic, or positive');
Check.IsTrue(nDestHeight.Value >= -1, 'Destination height must be -1 for source height, 0 for automatic, or positive');
END_METHOD

END_FUNCTION_BLOCK

// Nodes/Geometric and Coord Transform/Node_F_VN_RemapImageToPolarSpace
{attribute 'linkalways'} 
{attribute 'no_explicit_call' := 'This FB is a CLASS and must be accessed using methods or properties'}
{attribute 'enable_dynamic_creation'}
FUNCTION_BLOCK Node_F_VN_RemapImageToPolarSpace EXTENDS VisionNode
VAR
    ipSrcImage : _ITcVnImage;
    ipDestImage : _ITcVnImage;
    aCenter : _TcVnPoint2_REAL;
    hrPrev : _HRESULT(S_OK);
	hresult : _HRESULT(S_OK);
END_VAR

METHOD FB_init : BOOL
VAR_INPUT
	bInitRetains : BOOL; // if TRUE, the retain variables are initialized (warm start / cold start)
	bInCopyCode : BOOL;  // if TRUE, the instance afterwards gets moved into the copy code (online change)
END_VAR
AddInput('ipSrcImage', ipSrcImage);
AddInput('aCenter', aCenter);
AddInput('hrPrev', hrPrev);
AddOutput('ipDestImage', ipDestImage);
AddOutput('hresult',hresult);
END_METHOD

METHOD PUBLIC  Clone : I_Node
VAR
	pNode : POINTER TO Node_F_VN_RemapImageToPolarSpace;
END_VAR
pNode := __NEW(Node_F_VN_RemapImageToPolarSpace);
Clone := pNode^;
END_METHOD

METHOD PROTECTED OnExecute
hresult.Value := F_VN_RemapImageToPolarSpace(
    ipSrcImage := ipSrcImage.Value,
	ipDestImage := ipDestImage.Value,
    aCenter := aCenter.Value,
	hrPrev:= hrPrev.Value);
END_METHOD

METHOD PUBLIC PreExecutionCheck
VAR_INPUT
	Check : I_PreExecutionChecks;
END_VAR
Check.IsTrue(ipSrcImage.IsValid, 'ipSrcImage must contain an image');
END_METHOD

END_FUNCTION_BLOCK

// Nodes/Geometric and Coord Transform/Node_F_VN_RemapImageToPolarSpaceExp
{attribute 'linkalways'}
{attribute 'no_explicit_call' := 'This FB is a CLASS and must be accessed using methods or properties'}
{attribute 'enable_dynamic_creation'}
FUNCTION_BLOCK Node_F_VN_RemapImageToPolarSpaceExp EXTENDS VisionNode
VAR
    ipSrcImage : _ITcVnImage;
    ipDestImage : _ITcVnImage;
    aCenter : _TcVnPoint2_REAL;
    fMaxRadius : _LREAL(0);
    eInterpolationType : _ETcVnInterpolationType(ETcVnInterpolationType.TCVN_IT_BILINEAR);
    hrPrev : _HRESULT(S_OK);
    hresult : _HRESULT(S_OK);
END_VAR

METHOD FB_init : BOOL
VAR_INPUT
    bInitRetains : BOOL;
    bInCopyCode : BOOL;
END_VAR
AddInput('ipSrcImage', ipSrcImage);
AddOutput('ipDestImage', ipDestImage);
AddInput('aCenter', aCenter);
AddParameter('fMaxRadius', fMaxRadius);
AddParameter('eInterpolationType', eInterpolationType);
AddInput('hrPrev', hrPrev);
AddOutput('hresult', hresult);
END_METHOD

METHOD PUBLIC Clone : I_Node
VAR
    pNode : POINTER TO Node_F_VN_RemapImageToPolarSpaceExp;
END_VAR
pNode := __NEW(Node_F_VN_RemapImageToPolarSpaceExp);
Clone := pNode^;
END_METHOD

METHOD PROTECTED OnExecute
hresult.Value := F_VN_RemapImageToPolarSpaceExp(
    ipSrcImage := ipSrcImage.Value,
    ipDestImage := ipDestImage.Value,
    aCenter := aCenter.Value,
    fMaxRadius := fMaxRadius.Value,
    eInterpolationType := eInterpolationType.Value,
    hrPrev := hrPrev.Value);
END_METHOD

METHOD PUBLIC PreExecutionCheck
VAR_INPUT
    Check : I_PreExecutionChecks;
END_VAR
Check.IsTrue(ipSrcImage.IsValid, 'ipSrcImage must contain an image');
Check.IsTrue((ipDestImage.Value = 0) OR (ipDestImage.Value <> ipSrcImage.Value), 'Destination must be different from the source image');
Check.IsTrue((eInterpolationType.Value = ETcVnInterpolationType.TCVN_IT_NEAREST_NEIGHBOR) OR
             (eInterpolationType.Value = ETcVnInterpolationType.TCVN_IT_BILINEAR) OR
             (eInterpolationType.Value = ETcVnInterpolationType.TCVN_IT_BICUBIC) OR
             (eInterpolationType.Value = ETcVnInterpolationType.TCVN_IT_AREA_BASED) OR
             (eInterpolationType.Value = ETcVnInterpolationType.TCVN_IT_LANCZOS4), 'Unsupported eInterpolationType');
Check.IsTrue(fMaxRadius.Value >= 0.0, 'Maximum radius must be non-negative; zero selects it automatically');
END_METHOD

END_FUNCTION_BLOCK

// Nodes/Geometric and Coord Transform/Node_F_VN_RemapImageToPolarSpaceExp2
{attribute 'linkalways'}
{attribute 'no_explicit_call' := 'This FB is a CLASS and must be accessed using methods or properties'}
{attribute 'enable_dynamic_creation'}
FUNCTION_BLOCK Node_F_VN_RemapImageToPolarSpaceExp2 EXTENDS VisionNode
VAR
    ipSrcImage : _ITcVnImage;
    ipDestImage : _ITcVnImage;
    aCenter : _TcVnPoint2_REAL;
    fMaxRadius : _LREAL(0);
    eInterpolationType : _ETcVnInterpolationType(ETcVnInterpolationType.TCVN_IT_BILINEAR);
    nDestWidth : _DINT(-1);
    nDestHeight : _DINT(-1);
    hrPrev : _HRESULT(S_OK);
    hresult : _HRESULT(S_OK);
END_VAR

METHOD FB_init : BOOL
VAR_INPUT
    bInitRetains : BOOL;
    bInCopyCode : BOOL;
END_VAR
AddInput('ipSrcImage', ipSrcImage);
AddOutput('ipDestImage', ipDestImage);
AddInput('aCenter', aCenter);
AddParameter('fMaxRadius', fMaxRadius);
AddParameter('eInterpolationType', eInterpolationType);
AddParameter('nDestWidth', nDestWidth);
AddParameter('nDestHeight', nDestHeight);
AddInput('hrPrev', hrPrev);
AddOutput('hresult', hresult);
END_METHOD

METHOD PUBLIC Clone : I_Node
VAR
    pNode : POINTER TO Node_F_VN_RemapImageToPolarSpaceExp2;
END_VAR
pNode := __NEW(Node_F_VN_RemapImageToPolarSpaceExp2);
Clone := pNode^;
END_METHOD

METHOD PROTECTED OnExecute
hresult.Value := F_VN_RemapImageToPolarSpaceExp2(
    ipSrcImage := ipSrcImage.Value,
    ipDestImage := ipDestImage.Value,
    aCenter := aCenter.Value,
    fMaxRadius := fMaxRadius.Value,
    eInterpolationType := eInterpolationType.Value,
    nDestWidth := nDestWidth.Value,
    nDestHeight := nDestHeight.Value,
    hrPrev := hrPrev.Value);
END_METHOD

METHOD PUBLIC PreExecutionCheck
VAR_INPUT
    Check : I_PreExecutionChecks;
END_VAR
Check.IsTrue(ipSrcImage.IsValid, 'ipSrcImage must contain an image');
Check.IsTrue((ipDestImage.Value = 0) OR (ipDestImage.Value <> ipSrcImage.Value), 'Destination must be different from the source image');
Check.IsTrue((eInterpolationType.Value = ETcVnInterpolationType.TCVN_IT_NEAREST_NEIGHBOR) OR
             (eInterpolationType.Value = ETcVnInterpolationType.TCVN_IT_BILINEAR) OR
             (eInterpolationType.Value = ETcVnInterpolationType.TCVN_IT_BICUBIC) OR
             (eInterpolationType.Value = ETcVnInterpolationType.TCVN_IT_AREA_BASED) OR
             (eInterpolationType.Value = ETcVnInterpolationType.TCVN_IT_LANCZOS4), 'Unsupported eInterpolationType');
Check.IsTrue(fMaxRadius.Value >= 0.0, 'Maximum radius must be non-negative; zero selects it automatically');
Check.IsTrue(nDestWidth.Value >= -1, 'Destination width must be -1 for source width, 0 for automatic, or positive');
Check.IsTrue(nDestHeight.Value >= -1, 'Destination height must be -1 for source height, 0 for automatic, or positive');
END_METHOD

END_FUNCTION_BLOCK

// Nodes/Geometric and Coord Transform/Node_F_VN_ResizeImage
{attribute 'linkalways'} 
{attribute 'no_explicit_call' := 'This FB is a CLASS and must be accessed using methods or properties'}
{attribute 'enable_dynamic_creation'}
FUNCTION_BLOCK Node_F_VN_ResizeImage EXTENDS VisionNode
VAR
    ipSrcImage : _ITcVnImage;
    ipDestImage : _ITcVnImage;
    nWidth : _UDINT(0);
    nHeight : _UDINT(0);
    eInterpolationType : _ETcVnInterpolationType(ETcVnInterpolationType.TCVN_IT_NEAREST_NEIGHBOR);
    hrPrev : _HRESULT(S_OK);
	hresult : _HRESULT(S_OK);
END_VAR

METHOD FB_init : BOOL
VAR_INPUT
	bInitRetains : BOOL; // if TRUE, the retain variables are initialized (warm start / cold start)
	bInCopyCode : BOOL;  // if TRUE, the instance afterwards gets moved into the copy code (online change)
END_VAR
AddInput('ipSrcImage', ipSrcImage);
AddParameter('nWidth', nWidth);
AddParameter('nHeight', nHeight);
AddParameter('eInterpolationType', eInterpolationType);
AddInput('hrPrev', hrPrev);
AddOutput('ipDestImage', ipDestImage);
AddOutput('hresult',hresult);
END_METHOD

METHOD PUBLIC  Clone : I_Node
VAR
	pNode : POINTER TO Node_F_VN_ResizeImage;
END_VAR
pNode := __NEW(Node_F_VN_ResizeImage);
Clone := pNode^;
END_METHOD

METHOD PROTECTED OnExecute
hresult.Value := F_VN_ResizeImage(
    ipSrcImage := ipSrcImage.Value,
	ipDestImage := ipDestImage.Value,
    nWidth := nWidth.Value,
    nHeight := nHeight.Value,
    eInterpolationType := eInterpolationType.Value,
	hrPrev:= hrPrev.Value);
END_METHOD

METHOD PUBLIC PreExecutionCheck
VAR_INPUT
	Check : I_PreExecutionChecks;
END_VAR
Check.IsTrue(ipSrcImage.IsValid, 'ipSrcImage must contain an image');
END_METHOD

END_FUNCTION_BLOCK

// Nodes/Geometric and Coord Transform/Node_F_VN_ResizeImageExp
{attribute 'linkalways'} 
{attribute 'no_explicit_call' := 'This FB is a CLASS and must be accessed using methods or properties'}
{attribute 'enable_dynamic_creation'}
FUNCTION_BLOCK Node_F_VN_ResizeImageExp EXTENDS VisionNode
VAR
    ipSrcImage : _ITcVnImage;
    ipDestImage : _ITcVnImage;
    nWidth : _UDINT(0);
    nHeight : _UDINT(0);
    eInterpolationType : _ETcVnInterpolationType(ETcVnInterpolationType.TCVN_IT_NEAREST_NEIGHBOR);
    ePaddingMode : _ETcVnPaddingMode(ETcVnPaddingMode.TCVN_PM_NONE);
    aBorderValue : _TcVnVector4_LREAL;
    hrPrev : _HRESULT(S_OK);
	hresult : _HRESULT(S_OK);
END_VAR

METHOD FB_init : BOOL
VAR_INPUT
	bInitRetains : BOOL; // if TRUE, the retain variables are initialized (warm start / cold start)
	bInCopyCode : BOOL;  // if TRUE, the instance afterwards gets moved into the copy code (online change)
END_VAR
AddInput('ipSrcImage', ipSrcImage);
AddParameter('nWidth', nWidth);
AddParameter('nHeight', nHeight);
AddParameter('eInterpolationType', eInterpolationType);
AddParameter('ePaddingMode', ePaddingMode);
AddInput('aBorderValue', aBorderValue);
AddInput('hrPrev', hrPrev);
AddOutput('ipDestImage', ipDestImage);
AddOutput('hresult',hresult);
END_METHOD

METHOD PUBLIC  Clone : I_Node
VAR
	pNode : POINTER TO Node_F_VN_ResizeImageExp;
END_VAR
pNode := __NEW(Node_F_VN_ResizeImageExp);
Clone := pNode^;
END_METHOD

METHOD PROTECTED OnExecute
hresult.Value := F_VN_ResizeImageExp(
    ipSrcImage := ipSrcImage.Value,
	ipDestImage := ipDestImage.Value,
    nWidth := nWidth.Value,
    nHeight := nHeight.Value,
    eInterpolationType := eInterpolationType.Value,
    ePaddingMode := ePaddingMode.Value,
    aBorderValue := aBorderValue.Value,
	hrPrev:= hrPrev.Value);
END_METHOD

METHOD PUBLIC PreExecutionCheck
VAR_INPUT
	Check : I_PreExecutionChecks;
END_VAR
Check.IsTrue(ipSrcImage.IsValid, 'ipSrcImage must contain an image');
END_METHOD

END_FUNCTION_BLOCK

// Nodes/Geometric and Coord Transform/Node_F_VN_ResizeRegion_TcVnRectangle_DINT
{attribute 'linkalways'} 
{attribute 'no_explicit_call' := 'This FB is a CLASS and must be accessed using methods or properties'}
{attribute 'enable_dynamic_creation'}
FUNCTION_BLOCK Node_F_VN_ResizeRegion_TcVnRectangle_DINT EXTENDS VisionNode
VAR
	stSrcRect : _TcVnRectangle_DINT;
	stDestRect : _TcVnRectangle_DINT;
	fWidthRatio : _REAL(0);
	fHeightRatio : _REAL(0);
	nMinWidthOffset : _DINT(0);
	nMinHeightOffset : _DINT(0);
    ipImage : _ITcVnImage;
    hrPrev : _HRESULT(S_OK);
	hresult : _HRESULT(S_OK);
END_VAR

METHOD FB_init : BOOL
VAR_INPUT
	bInitRetains : BOOL; // if TRUE, the retain variables are initialized (warm start / cold start)
	bInCopyCode : BOOL;  // if TRUE, the instance afterwards gets moved into the copy code (online change)
END_VAR
AddInput('stSrcRect', stSrcRect);
AddInput('ipImage', ipImage);
AddInput('hrPrev', hrPrev);
AddParameter('fWidthRatio', fWidthRatio);
AddParameter('fHeightRatio', fHeightRatio);
AddParameter('nMinWidthOffset', nMinWidthOffset);
AddParameter('nMinHeightOffset', nMinHeightOffset);
AddOutput('stDestRect', stDestRect);
AddOutput('hresult',hresult);
END_METHOD

METHOD PUBLIC  Clone : I_Node
VAR
	pNode : POINTER TO Node_F_VN_ResizeRegion_TcVnRectangle_DINT;
END_VAR
pNode := __NEW(Node_F_VN_ResizeRegion_TcVnRectangle_DINT);
Clone := pNode^;
END_METHOD

METHOD PROTECTED OnExecute
hresult.Value := F_VN_ResizeRegion_TcVnRectangle_DINT(
    stSrcRect := stSrcRect.Value,
	stDestRect := stDestRect.Value,
	fWidthRatio := fWidthRatio.Value,
	fHeightRatio := fHeightRatio.Value,
	nMinWidthOffset := nMinWidthOffset.Value,
	nMinHeightOffset := nMinHeightOffset.Value,
	ipImage := ipImage.Value,
	hrPrev:= hrPrev.Value);
END_METHOD

METHOD PUBLIC PreExecutionCheck
VAR_INPUT
	Check : I_PreExecutionChecks;
END_VAR
END_METHOD

END_FUNCTION_BLOCK

// Nodes/Geometric and Coord Transform/Node_F_VN_RotateImage
{attribute 'linkalways'} 
{attribute 'no_explicit_call' := 'This FB is a CLASS and must be accessed using methods or properties'}
{attribute 'enable_dynamic_creation'}
FUNCTION_BLOCK Node_F_VN_RotateImage EXTENDS VisionNode
VAR
    ipSrcImage : _ITcVnImage;
    ipDestImage : _ITcVnImage;
    eAngle : _ETcVnRotationAngle(ETcVnRotationAngle.TCVN_RA_90_DEG);
    hrPrev : _HRESULT(S_OK);
	hresult : _HRESULT(S_OK);
END_VAR

METHOD FB_init : BOOL
VAR_INPUT
	bInitRetains : BOOL; // if TRUE, the retain variables are initialized (warm start / cold start)
	bInCopyCode : BOOL;  // if TRUE, the instance afterwards gets moved into the copy code (online change)
END_VAR
AddInput('ipSrcImage', ipSrcImage);
AddParameter('eAngle', eAngle);
AddInput('hrPrev', hrPrev);
AddOutput('ipDestImage', ipDestImage);
AddOutput('hresult',hresult);
END_METHOD

METHOD PUBLIC  Clone : I_Node
VAR
	pNode : POINTER TO Node_F_VN_RotateImage;
END_VAR
pNode := __NEW(Node_F_VN_RotateImage);
Clone := pNode^;
END_METHOD

METHOD PROTECTED OnExecute
hresult.Value := F_VN_RotateImage(
    ipSrcImage := ipSrcImage.Value,
	ipDestImage := ipDestImage.Value,
    eAngle := eAngle.Value,
	hrPrev:= hrPrev.Value);
END_METHOD

METHOD PUBLIC PreExecutionCheck
VAR_INPUT
	Check : I_PreExecutionChecks;
END_VAR
Check.IsTrue(ipSrcImage.IsValid, 'ipSrcImage must contain an image');
END_METHOD

END_FUNCTION_BLOCK

// Nodes/Geometric and Coord Transform/Node_F_VN_RotateImageExp
{attribute 'linkalways'} 
{attribute 'no_explicit_call' := 'This FB is a CLASS and must be accessed using methods or properties'}
{attribute 'enable_dynamic_creation'}
FUNCTION_BLOCK Node_F_VN_RotateImageExp EXTENDS VisionNode
VAR
    ipSrcImage : _ITcVnImage;
    ipDestImage : _ITcVnImage;
    fAngleDeg : _LREAL(0.0);
    bAdjustDestSize : _BOOL(FALSE);
    hrPrev : _HRESULT(S_OK);
	hresult : _HRESULT(S_OK);
END_VAR

METHOD FB_init : BOOL
VAR_INPUT
	bInitRetains : BOOL; // if TRUE, the retain variables are initialized (warm start / cold start)
	bInCopyCode : BOOL;  // if TRUE, the instance afterwards gets moved into the copy code (online change)
END_VAR
AddInput('ipSrcImage', ipSrcImage);
AddParameter('fAngleDeg', fAngleDeg);
AddParameter('bAdjustDestSize', bAdjustDestSize);
AddInput('hrPrev', hrPrev);
AddOutput('ipDestImage', ipDestImage);
AddOutput('hresult',hresult);
END_METHOD

METHOD PUBLIC  Clone : I_Node
VAR
	pNode : POINTER TO Node_F_VN_RotateImageExp;
END_VAR
pNode := __NEW(Node_F_VN_RotateImageExp);
Clone := pNode^;
END_METHOD

METHOD PROTECTED OnExecute
hresult.Value := F_VN_RotateImageExp(
    ipSrcImage := ipSrcImage.Value,
	ipDestImage := ipDestImage.Value,
    fAngleDeg := fAngleDeg.Value,
    bAdjustDestSize := bAdjustDestSize.Value,
	hrPrev:= hrPrev.Value);
END_METHOD

METHOD PUBLIC PreExecutionCheck
VAR_INPUT
	Check : I_PreExecutionChecks;
END_VAR
Check.IsTrue(ipSrcImage.IsValid, 'ipSrcImage must contain an image');
END_METHOD

END_FUNCTION_BLOCK

// Nodes/Geometric and Coord Transform/Node_F_VN_RotateImageExp2
{attribute 'linkalways'} 
{attribute 'no_explicit_call' := 'This FB is a CLASS and must be accessed using methods or properties'}
{attribute 'enable_dynamic_creation'}
FUNCTION_BLOCK Node_F_VN_RotateImageExp2 EXTENDS VisionNode
VAR
    ipSrcImage : _ITcVnImage;
    ipDestImage : _ITcVnImage;
    fAngleDeg : _LREAL(0.0);
    bAdjustDestSize : _BOOL(FALSE);
    eInterpolationType : _ETcVnInterpolationType(ETcVnInterpolationType.TCVN_IT_NEAREST_NEIGHBOR);
    eBorderInterpolation : 	_ETcVnBorderInterpolationMethod(ETcVnBorderInterpolationMethod.TCVN_BIM_DEFAULT);
    aBorderValue : _TcVnVector4_LREAL;
    hrPrev : _HRESULT(S_OK);
	hresult : _HRESULT(S_OK);
END_VAR

METHOD FB_init : BOOL
VAR_INPUT
	bInitRetains : BOOL; // if TRUE, the retain variables are initialized (warm start / cold start)
	bInCopyCode : BOOL;  // if TRUE, the instance afterwards gets moved into the copy code (online change)
END_VAR
AddInput('ipSrcImage', ipSrcImage);
AddParameter('fAngleDeg', fAngleDeg);
AddParameter('bAdjustDestSize', bAdjustDestSize);
AddParameter('eInterpolationType', eInterpolationType);
AddParameter('eBorderInterpolation', eBorderInterpolation);
AddInput('aBorderValue', aBorderValue);
AddInput('hrPrev', hrPrev);
AddOutput('ipDestImage', ipDestImage);
AddOutput('hresult',hresult);
END_METHOD

METHOD PUBLIC  Clone : I_Node
VAR
	pNode : POINTER TO Node_F_VN_RotateImageExp2;
END_VAR
pNode := __NEW(Node_F_VN_RotateImageExp2);
Clone := pNode^;
END_METHOD

METHOD PROTECTED OnExecute
hresult.Value := F_VN_RotateImageExp2(
    ipSrcImage := ipSrcImage.Value,
	ipDestImage := ipDestImage.Value,
    fAngleDeg := fAngleDeg.Value,
    bAdjustDestSize := bAdjustDestSize.Value,
    eInterpolationType := eInterpolationType.Value,
    eBorderInterpolation := eBorderInterpolation.Value,
    aBorderValue := aBorderValue.Value,
	hrPrev:= hrPrev.Value);
END_METHOD

METHOD PUBLIC PreExecutionCheck
VAR_INPUT
	Check : I_PreExecutionChecks;
END_VAR
Check.IsTrue(ipSrcImage.IsValid, 'ipSrcImage must contain an image');
END_METHOD

END_FUNCTION_BLOCK

// Nodes/Geometric and Coord Transform/Node_F_VN_WarpAffine
{attribute 'linkalways'} 
{attribute 'no_explicit_call' := 'This FB is a CLASS and must be accessed using methods or properties'}
{attribute 'enable_dynamic_creation'}
FUNCTION_BLOCK Node_F_VN_WarpAffine EXTENDS VisionNode
VAR
	ipSrcImage : _ITcVnImage;
    ipDestImage : _ITcVnImage;
    aTransformationMatrix : _TcVnMatrix2x3_LREAL;
    hrPrev : _HRESULT(S_OK);
	hresult : _HRESULT(S_OK);
END_VAR

METHOD FB_init : BOOL
VAR_INPUT
	bInitRetains : BOOL; // if TRUE, the retain variables are initialized (warm start / cold start)
	bInCopyCode : BOOL;  // if TRUE, the instance afterwards gets moved into the copy code (online change)
END_VAR
AddInput('ipSrcImage', ipSrcImage);
AddInput('aTransformationMatrix', aTransformationMatrix);
AddInput('hrPrev', hrPrev);
AddOutput('ipDestImage', ipDestImage);
AddOutput('hresult',hresult);
END_METHOD

METHOD PUBLIC  Clone : I_Node
VAR
	pNode : POINTER TO Node_F_VN_WarpAffine;
END_VAR
pNode := __NEW(Node_F_VN_WarpAffine);
Clone := pNode^;
END_METHOD

METHOD PROTECTED OnExecute
hresult.Value := F_VN_WarpAffine(
	ipSrcImage := ipSrcImage.Value, 
	ipDestImage := ipDestImage.Value, 
	aTransformationMatrix := aTransformationMatrix.Value, 
	hrPrev := hrPrev.Value);
END_METHOD

METHOD PUBLIC PreExecutionCheck
VAR_INPUT
	Check : I_PreExecutionChecks;
END_VAR
Check.IsTrue(ipSrcImage.IsValid, 'ipSrcImage must contain an image');
END_METHOD

END_FUNCTION_BLOCK

// Nodes/Geometric and Coord Transform/Node_F_VN_WarpAffine_Container
{attribute 'linkalways'} 
{attribute 'no_explicit_call' := 'This FB is a CLASS and must be accessed using methods or properties'}
{attribute 'enable_dynamic_creation'}
FUNCTION_BLOCK Node_F_VN_WarpAffine_Container EXTENDS VisionNode
VAR
	ipSrcPoints : _ITcVnContainer;
    ipDestPoints : _ITcVnContainer;
    aTransformationMatrix : _TcVnMatrix2x3_LREAL;
    hrPrev : _HRESULT(S_OK);
	hresult : _HRESULT(S_OK);
END_VAR

METHOD FB_init : BOOL
VAR_INPUT
	bInitRetains : BOOL; // if TRUE, the retain variables are initialized (warm start / cold start)
	bInCopyCode : BOOL;  // if TRUE, the instance afterwards gets moved into the copy code (online change)
END_VAR
AddInput('ipSrcPoints', ipSrcPoints);
AddInput('aTransformationMatrix', aTransformationMatrix);
AddInput('hrPrev', hrPrev);
AddOutput('ipDestPoints', ipDestPoints);
AddOutput('hresult',hresult);
END_METHOD

METHOD PUBLIC  Clone : I_Node
VAR
	pNode : POINTER TO Node_F_VN_WarpAffine_Container;
END_VAR
pNode := __NEW(Node_F_VN_WarpAffine_Container);
Clone := pNode^;
END_METHOD

METHOD PROTECTED OnExecute
hresult.Value := F_VN_WarpAffine_Container(
	ipSrcPoints := ipSrcPoints.Value, 
	ipDestPoints := ipDestPoints.Value, 
	aTransformationMatrix := aTransformationMatrix.Value, 
	hrPrev := hrPrev.Value);
END_METHOD

METHOD PUBLIC PreExecutionCheck
VAR_INPUT
	Check : I_PreExecutionChecks;
END_VAR
Check.IsTrue(ipSrcPoints.IsValid, 'ipSrcPoints must be a valid container');
Check.IsTrue((ipSrcPoints.IsType(TC_GLOBAL_CONST_LIST.ContainerType_Vector_TcVnPoint2_DINT) OR
              ipSrcPoints.IsType(TC_GLOBAL_CONST_LIST.ContainerType_Vector_TcVnPoint2_REAL) OR
              ipSrcPoints.IsType(TC_GLOBAL_CONST_LIST.ContainerType_Vector_TcVnPoint2_LREAL)),
              'ipSrcPoints contains incorrect type');
END_METHOD

END_FUNCTION_BLOCK

// Nodes/Geometric and Coord Transform/Node_F_VN_WarpAffine_Point
{attribute 'linkalways'} 
{attribute 'no_explicit_call' := 'This FB is a CLASS and must be accessed using methods or properties'}
{attribute 'enable_dynamic_creation'}
FUNCTION_BLOCK Node_F_VN_WarpAffine_Point EXTENDS VisionNode
VAR
	aSrcPoint : _TcVnPoint2_LREAL;
    aDestPoint : _TcVnPoint2_LREAL;
    aTransformationMatrix : _TcVnMatrix2x3_LREAL;
    hrPrev : _HRESULT(S_OK);
	hresult : _HRESULT(S_OK);
END_VAR

METHOD FB_init : BOOL
VAR_INPUT
	bInitRetains : BOOL; // if TRUE, the retain variables are initialized (warm start / cold start)
	bInCopyCode : BOOL;  // if TRUE, the instance afterwards gets moved into the copy code (online change)
END_VAR
AddInput('aSrcPoint', aSrcPoint);
AddInput('aTransformationMatrix', aTransformationMatrix);
AddInput('hrPrev', hrPrev);
AddOutput('aDestPoint', aDestPoint);
AddOutput('hresult',hresult);
END_METHOD

METHOD PUBLIC  Clone : I_Node
VAR
	pNode : POINTER TO Node_F_VN_WarpAffine_Point;
END_VAR
pNode := __NEW(Node_F_VN_WarpAffine_Point);
Clone := pNode^;
END_METHOD

METHOD PROTECTED OnExecute
hresult.Value := F_VN_WarpAffine_Point(
	aSrcPoint := aSrcPoint.Value, 
	aDestPoint := aDestPoint.Value, 
	aTransformationMatrix := aTransformationMatrix.Value, 
	hrPrev := hrPrev.Value);
END_METHOD

METHOD PUBLIC PreExecutionCheck
VAR_INPUT
	Check : I_PreExecutionChecks;
END_VAR
END_METHOD

END_FUNCTION_BLOCK

// Nodes/Geometric and Coord Transform/Node_F_VN_WarpAffine_Rectangle
{attribute 'linkalways'} 
{attribute 'no_explicit_call' := 'This FB is a CLASS and must be accessed using methods or properties'}
{attribute 'enable_dynamic_creation'}
FUNCTION_BLOCK Node_F_VN_WarpAffine_Rectangle EXTENDS VisionNode
VAR
	nTopLeftX : _UDINT(0);
    nTopLeftY : _UDINT(0);
    nBottomRightX : _UDINT(0);
    nBottomRightY : _UDINT(0);
    ipDestPoints : _ITcVnContainer;
    aTransformationMatrix : _TcVnMatrix2x3_LREAL;
    hrPrev : _HRESULT(S_OK);
	hresult : _HRESULT(S_OK);
END_VAR

METHOD FB_init : BOOL
VAR_INPUT
	bInitRetains : BOOL; // if TRUE, the retain variables are initialized (warm start / cold start)
	bInCopyCode : BOOL;  // if TRUE, the instance afterwards gets moved into the copy code (online change)
END_VAR
AddParameter('nTopLeftX', nTopLeftX);
AddParameter('nTopLeftY', nTopLeftY);
AddParameter('nBottomRightX', nBottomRightX);
AddParameter('nBottomRightY', nBottomRightY);
AddInput('aTransformationMatrix', aTransformationMatrix);
AddInput('hrPrev', hrPrev);
AddOutput('ipDestPoints', ipDestPoints);
AddOutput('hresult',hresult);
END_METHOD

METHOD PUBLIC  Clone : I_Node
VAR
	pNode : POINTER TO Node_F_VN_WarpAffine_Rectangle;
END_VAR
pNode := __NEW(Node_F_VN_WarpAffine_Rectangle);
Clone := pNode^;
END_METHOD

METHOD PROTECTED OnExecute
hresult.Value := F_VN_WarpAffine_Rectangle(
	nTopLeftX := nTopLeftX.Value,
    nTopLeftY := nTopLeftY.Value,
    nBottomRightX := nBottomRightX.Value,
    nBottomRightY := nBottomRightY.Value,
	ipDestPoints := ipDestPoints.Value, 
	aTransformationMatrix := aTransformationMatrix.Value, 
	hrPrev := hrPrev.Value);
END_METHOD

METHOD PUBLIC PreExecutionCheck
VAR_INPUT
	Check : I_PreExecutionChecks;
END_VAR
END_METHOD

END_FUNCTION_BLOCK

// Nodes/Geometric and Coord Transform/Node_F_VN_WarpAffineExp
{attribute 'linkalways'} 
{attribute 'no_explicit_call' := 'This FB is a CLASS and must be accessed using methods or properties'}
{attribute 'enable_dynamic_creation'}
FUNCTION_BLOCK Node_F_VN_WarpAffineExp EXTENDS VisionNode
VAR
	ipSrcImage : _ITcVnImage;
    ipDestImage : _ITcVnImage;
    aTransformationMatrix : _TcVnMatrix2x3_LREAL;
    nDestWidth : _UDINT(1);
    nDestHeight : _UDINT(1);
    eInterpolationType : _ETcVnInterpolationType(ETcVnInterpolationType.TCVN_IT_NEAREST_NEIGHBOR);
    bWarpInverse : _BOOL(FALSE);
    eBorderInterpolation : _ETcVnBorderInterpolationMethod(ETcVnBorderInterpolationMethod.TCVN_BIM_DEFAULT);
    fBorderValue : _LREAL(0.0);
    hrPrev : _HRESULT(S_OK);
	hresult : _HRESULT(S_OK);
END_VAR

METHOD FB_init : BOOL
VAR_INPUT
	bInitRetains : BOOL; // if TRUE, the retain variables are initialized (warm start / cold start)
	bInCopyCode : BOOL;  // if TRUE, the instance afterwards gets moved into the copy code (online change)
END_VAR
AddInput('ipSrcImage', ipSrcImage);
AddInput('aTransformationMatrix', aTransformationMatrix);
AddParameter('nDestWidth', nDestWidth);
AddParameter('nDestHeight', nDestHeight);
AddParameter('eInterpolationType', eInterpolationType);
AddParameter('bWarpInverse', bWarpInverse);
AddParameter('eBorderInterpolation', eBorderInterpolation);
AddParameter('fBorderValue', fBorderValue);
AddInput('hrPrev', hrPrev);
AddOutput('ipDestImage', ipDestImage);
AddOutput('hresult',hresult);
END_METHOD

METHOD PUBLIC  Clone : I_Node
VAR
	pNode : POINTER TO Node_F_VN_WarpAffineExp;
END_VAR
pNode := __NEW(Node_F_VN_WarpAffineExp);
Clone := pNode^;
END_METHOD

METHOD PROTECTED OnExecute
hresult.Value := F_VN_WarpAffineExp(
	ipSrcImage := ipSrcImage.Value,
	ipDestImage := ipDestImage.Value,
	aTransformationMatrix := aTransformationMatrix.Value,
    nDestWidth := nDestWidth.Value,
    nDestHeight := nDestHeight.Value,
    eInterpolationType := eInterpolationType.Value,
    bWarpInverse := bWarpInverse.Value,
    eBorderInterpolation := eBorderInterpolation.Value,
    fBorderValue := fBorderValue.Value,
	hrPrev := hrPrev.Value);
END_METHOD

METHOD PUBLIC PreExecutionCheck
VAR_INPUT
	Check : I_PreExecutionChecks;
END_VAR
VAR
    borderInterpolationMethodIsValid : BOOL;
END_VAR
Check.IsTrue(ipSrcImage.IsValid, 'ipSrcImage must contain an image');
Check.IsTrue(nDestWidth.Value > 0, 'nDestWidth must be greater than 0');
Check.IsTrue(nDestHeight.Value > 0, 'nDestHeight must be greater than 0');

CASE eBorderInterpolation.Value OF
    ETcVnBorderInterpolationMethod.TCVN_BIM_CONSTANT,
    ETcVnBorderInterpolationMethod.TCVN_BIM_REPLICATE,
    ETcVnBorderInterpolationMethod.TCVN_BIM_REFLECT,
    ETcVnBorderInterpolationMethod.TCVN_BIM_WRAP,
    ETcVnBorderInterpolationMethod.TCVN_BIM_REFLECT_101,
    //ETcVnBorderInterpolationMethod.TCVN_BIM_DEFAULT, // Same as REFLECT_101
    ETcVnBorderInterpolationMethod.TCVN_BIM_TRANSPARENT :
        borderInterpolationMethodIsValid := TRUE;
END_CASE

Check.IsTrue(borderInterpolationMethodIsValid, 'eBorderInterpolation ISOLATED not supported');
END_METHOD

END_FUNCTION_BLOCK

// Nodes/Geometric and Coord Transform/Node_F_VN_WarpPerspective
{attribute 'linkalways'} 
{attribute 'no_explicit_call' := 'This FB is a CLASS and must be accessed using methods or properties'}
{attribute 'enable_dynamic_creation'}
FUNCTION_BLOCK Node_F_VN_WarpPerspective EXTENDS VisionNode
VAR
	ipSrcImage : _ITcVnImage;
    ipDestImage : _ITcVnImage;
    aTransformationMatrix : _TcVnMatrix3x3_LREAL;
    hrPrev : _HRESULT(S_OK);
	hresult : _HRESULT(S_OK);
END_VAR

METHOD FB_init : BOOL
VAR_INPUT
	bInitRetains : BOOL; // if TRUE, the retain variables are initialized (warm start / cold start)
	bInCopyCode : BOOL;  // if TRUE, the instance afterwards gets moved into the copy code (online change)
END_VAR
AddInput('ipSrcImage', ipSrcImage);
AddInput('aTransformationMatrix', aTransformationMatrix);
AddInput('hrPrev', hrPrev);
AddOutput('ipDestImage', ipDestImage);
AddOutput('hresult',hresult);
END_METHOD

METHOD PUBLIC  Clone : I_Node
VAR
	pNode : POINTER TO Node_F_VN_WarpPerspective;
END_VAR
pNode := __NEW(Node_F_VN_WarpPerspective);
Clone := pNode^;
END_METHOD

METHOD PROTECTED OnExecute
hresult.Value := F_VN_WarpPerspective(
	ipSrcImage := ipSrcImage.Value, 
	ipDestImage := ipDestImage.Value, 
	aTransformationMatrix := aTransformationMatrix.Value, 
	hrPrev := hrPrev.Value);
END_METHOD

METHOD PUBLIC PreExecutionCheck
VAR_INPUT
	Check : I_PreExecutionChecks;
END_VAR
Check.IsTrue(ipSrcImage.IsValid, 'ipSrcImage must contain an image');
END_METHOD

END_FUNCTION_BLOCK

// Nodes/Geometric and Coord Transform/Node_F_VN_WarpPerspective_Container
{attribute 'linkalways'} 
{attribute 'no_explicit_call' := 'This FB is a CLASS and must be accessed using methods or properties'}
{attribute 'enable_dynamic_creation'}
FUNCTION_BLOCK Node_F_VN_WarpPerspective_Container EXTENDS VisionNode
VAR
	ipSrcPoints : _ITcVnContainer;
    ipDestPoints : _ITcVnContainer;
    aTransformationMatrix : _TcVnMatrix3x3_LREAL;
    hrPrev : _HRESULT(S_OK);
	hresult : _HRESULT(S_OK);
END_VAR

METHOD FB_init : BOOL
VAR_INPUT
	bInitRetains : BOOL; // if TRUE, the retain variables are initialized (warm start / cold start)
	bInCopyCode : BOOL;  // if TRUE, the instance afterwards gets moved into the copy code (online change)
END_VAR
AddInput('ipSrcPoints', ipSrcPoints);
AddInput('aTransformationMatrix', aTransformationMatrix);
AddInput('hrPrev', hrPrev);
AddOutput('ipDestPoints', ipDestPoints);
AddOutput('hresult',hresult);
END_METHOD

METHOD PUBLIC  Clone : I_Node
VAR
	pNode : POINTER TO Node_F_VN_WarpPerspective_Container;
END_VAR
pNode := __NEW(Node_F_VN_WarpPerspective_Container);
Clone := pNode^;
END_METHOD

METHOD PROTECTED OnExecute
hresult.Value := F_VN_WarpPerspective_Container(
	ipSrcPoints := ipSrcPoints.Value, 
	ipDestPoints := ipDestPoints.Value, 
	aTransformationMatrix := aTransformationMatrix.Value, 
	hrPrev := hrPrev.Value);
END_METHOD

METHOD PUBLIC PreExecutionCheck
VAR_INPUT
	Check : I_PreExecutionChecks;
END_VAR
Check.IsTrue(ipSrcPoints.IsValid, 'ipSrcPoints must be a valid container');
Check.IsTrue((ipSrcPoints.IsType(TC_GLOBAL_CONST_LIST.ContainerType_Vector_TcVnPoint2_DINT) OR
              ipSrcPoints.IsType(TC_GLOBAL_CONST_LIST.ContainerType_Vector_TcVnPoint2_REAL) OR
              ipSrcPoints.IsType(TC_GLOBAL_CONST_LIST.ContainerType_Vector_TcVnPoint2_LREAL)),
              'ipSrcPoints contains incorrect type');
END_METHOD

END_FUNCTION_BLOCK

// Nodes/Geometric and Coord Transform/Node_F_VN_WarpPerspective_Point
{attribute 'linkalways'} 
{attribute 'no_explicit_call' := 'This FB is a CLASS and must be accessed using methods or properties'}
{attribute 'enable_dynamic_creation'}
FUNCTION_BLOCK Node_F_VN_WarpPerspective_Point EXTENDS VisionNode
VAR
	aSrcPoint : _TcVnPoint2_LREAL;
    aDestPoint : _TcVnPoint2_LREAL;
    aTransformationMatrix : _TcVnMatrix3x3_LREAL;
    hrPrev : _HRESULT(S_OK);
	hresult : _HRESULT(S_OK);
END_VAR

METHOD FB_init : BOOL
VAR_INPUT
	bInitRetains : BOOL; // if TRUE, the retain variables are initialized (warm start / cold start)
	bInCopyCode : BOOL;  // if TRUE, the instance afterwards gets moved into the copy code (online change)
END_VAR
AddInput('aSrcPoint', aSrcPoint);
AddInput('aTransformationMatrix', aTransformationMatrix);
AddInput('hrPrev', hrPrev);
AddOutput('aDestPoint', aDestPoint);
AddOutput('hresult',hresult);
END_METHOD

METHOD PUBLIC  Clone : I_Node
VAR
	pNode : POINTER TO Node_F_VN_WarpPerspective_Point;
END_VAR
pNode := __NEW(Node_F_VN_WarpPerspective_Point);
Clone := pNode^;
END_METHOD

METHOD PROTECTED OnExecute
hresult.Value := F_VN_WarpPerspective_Point(
	aSrcPoint := aSrcPoint.Value, 
	aDestPoint := aDestPoint.Value, 
	aTransformationMatrix := aTransformationMatrix.Value, 
	hrPrev := hrPrev.Value);
END_METHOD

METHOD PUBLIC PreExecutionCheck
VAR_INPUT
	Check : I_PreExecutionChecks;
END_VAR
END_METHOD

END_FUNCTION_BLOCK

// Nodes/Geometric and Coord Transform/Node_F_VN_WarpPerspective_Rectangle
{attribute 'linkalways'} 
{attribute 'no_explicit_call' := 'This FB is a CLASS and must be accessed using methods or properties'}
{attribute 'enable_dynamic_creation'}
FUNCTION_BLOCK Node_F_VN_WarpPerspective_Rectangle EXTENDS VisionNode
VAR
	nTopLeftX : _UDINT(0);
    nTopLeftY : _UDINT(0);
    nBottomRightX : _UDINT(0);
    nBottomRightY : _UDINT(0);
    ipDestPoints : _ITcVnContainer;
    aTransformationMatrix : _TcVnMatrix3x3_LREAL;
    hrPrev : _HRESULT(S_OK);
	hresult : _HRESULT(S_OK);
END_VAR

METHOD FB_init : BOOL
VAR_INPUT
	bInitRetains : BOOL; // if TRUE, the retain variables are initialized (warm start / cold start)
	bInCopyCode : BOOL;  // if TRUE, the instance afterwards gets moved into the copy code (online change)
END_VAR
AddParameter('nTopLeftX', nTopLeftX);
AddParameter('nTopLeftY', nTopLeftY);
AddParameter('nBottomRightX', nBottomRightX);
AddParameter('nBottomRightY', nBottomRightY);
AddInput('aTransformationMatrix', aTransformationMatrix);
AddInput('hrPrev', hrPrev);
AddOutput('ipDestPoints', ipDestPoints);
AddOutput('hresult',hresult);
END_METHOD

METHOD PUBLIC  Clone : I_Node
VAR
	pNode : POINTER TO Node_F_VN_WarpPerspective_Rectangle;
END_VAR
pNode := __NEW(Node_F_VN_WarpPerspective_Rectangle);
Clone := pNode^;
END_METHOD

METHOD PROTECTED OnExecute
hresult.Value := F_VN_WarpPerspective_Rectangle(
	nTopLeftX := nTopLeftX.Value,
    nTopLeftY := nTopLeftY.Value,
    nBottomRightX := nBottomRightX.Value,
    nBottomRightY := nBottomRightY.Value,
	ipDestPoints := ipDestPoints.Value, 
	aTransformationMatrix := aTransformationMatrix.Value, 
	hrPrev := hrPrev.Value);
END_METHOD

METHOD PUBLIC PreExecutionCheck
VAR_INPUT
	Check : I_PreExecutionChecks;
END_VAR
END_METHOD

END_FUNCTION_BLOCK

// Nodes/Geometric and Coord Transform/Node_F_VN_WarpPerspectiveExp
{attribute 'linkalways'} 
{attribute 'no_explicit_call' := 'This FB is a CLASS and must be accessed using methods or properties'}
{attribute 'enable_dynamic_creation'}
FUNCTION_BLOCK Node_F_VN_WarpPerspectiveExp EXTENDS VisionNode
VAR
	ipSrcImage : _ITcVnImage;
    ipDestImage : _ITcVnImage;
    aTransformationMatrix : _TcVnMatrix3x3_LREAL;
    nDestWidth : _UDINT(1);
    nDestHeight : _UDINT(1);
    eInterpolationType : _ETcVnInterpolationType(ETcVnInterpolationType.TCVN_IT_NEAREST_NEIGHBOR);
    bWarpInverse : _BOOL(FALSE);
    eBorderInterpolation : _ETcVnBorderInterpolationMethod(ETcVnBorderInterpolationMethod.TCVN_BIM_DEFAULT);
    fBorderValue : _LREAL(0.0);
    hrPrev : _HRESULT(S_OK);
	hresult : _HRESULT(S_OK);
END_VAR

METHOD FB_init : BOOL
VAR_INPUT
	bInitRetains : BOOL; // if TRUE, the retain variables are initialized (warm start / cold start)
	bInCopyCode : BOOL;  // if TRUE, the instance afterwards gets moved into the copy code (online change)
END_VAR
AddInput('ipSrcImage', ipSrcImage);
AddInput('aTransformationMatrix', aTransformationMatrix);
AddParameter('nDestWidth', nDestWidth);
AddParameter('nDestHeight', nDestHeight);
AddParameter('eInterpolationType', eInterpolationType);
AddParameter('bWarpInverse', bWarpInverse);
AddParameter('eBorderInterpolation', eBorderInterpolation);
AddParameter('fBorderValue', fBorderValue);
AddInput('hrPrev', hrPrev);
AddOutput('ipDestImage', ipDestImage);
AddOutput('hresult',hresult);
END_METHOD

METHOD PUBLIC  Clone : I_Node
VAR
	pNode : POINTER TO Node_F_VN_WarpPerspectiveExp;
END_VAR
pNode := __NEW(Node_F_VN_WarpPerspectiveExp);
Clone := pNode^;
END_METHOD

METHOD PROTECTED OnExecute
hresult.Value := F_VN_WarpPerspectiveExp(
	ipSrcImage := ipSrcImage.Value,
	ipDestImage := ipDestImage.Value,
	aTransformationMatrix := aTransformationMatrix.Value,
    nDestWidth := nDestWidth.Value,
    nDestHeight := nDestHeight.Value,
    eInterpolationType := eInterpolationType.Value,
    bWarpInverse := bWarpInverse.Value,
    eBorderInterpolation := eBorderInterpolation.Value,
    fBorderValue := fBorderValue.Value,
	hrPrev := hrPrev.Value);
END_METHOD

METHOD PUBLIC PreExecutionCheck
VAR_INPUT
	Check : I_PreExecutionChecks;
END_VAR
VAR
    borderInterpolationMethodIsValid : BOOL;
END_VAR
Check.IsTrue(ipSrcImage.IsValid, 'ipSrcImage must contain an image');
Check.IsTrue(nDestWidth.Value > 0, 'nDestWidth must be greater than 0');
Check.IsTrue(nDestHeight.Value > 0, 'nDestHeight must be greater than 0');

CASE eBorderInterpolation.Value OF
    ETcVnBorderInterpolationMethod.TCVN_BIM_CONSTANT,
    ETcVnBorderInterpolationMethod.TCVN_BIM_REPLICATE,
    ETcVnBorderInterpolationMethod.TCVN_BIM_REFLECT,
    ETcVnBorderInterpolationMethod.TCVN_BIM_WRAP,
    ETcVnBorderInterpolationMethod.TCVN_BIM_REFLECT_101,
    //ETcVnBorderInterpolationMethod.TCVN_BIM_DEFAULT, // Same as REFLECT_101
    ETcVnBorderInterpolationMethod.TCVN_BIM_TRANSPARENT :
        borderInterpolationMethodIsValid := TRUE;
END_CASE

Check.IsTrue(borderInterpolationMethodIsValid, 'eBorderInterpolation ISOLATED not supported');
END_METHOD

END_FUNCTION_BLOCK

// Nodes/Helpers/Node_Mux10Way_ITcVnImage
{attribute 'linkalways'} 
{attribute 'no_explicit_call' := 'This FB is a CLASS and must be accessed using methods or properties'}
{attribute 'enable_dynamic_creation'}
FUNCTION_BLOCK Node_Mux10Way_ITcVnImage EXTENDS Node
VAR
	in0 : _ITcVnImage;
	in1 : _ITcVnImage;
	in2 : _ITcVnImage;
	in3 : _ITcVnImage;
	in4 : _ITcVnImage;
	in5 : _ITcVnImage;
	in6 : _ITcVnImage;
	in7 : _ITcVnImage;
	in8 : _ITcVnImage;
	in9 : _ITcVnImage;
	index : _BYTE(0);
    out : _ITcVnImage;
END_VAR

METHOD FB_init : BOOL
VAR_INPUT
	bInitRetains : BOOL; // if TRUE, the retain variables are initialized (warm start / cold start)
	bInCopyCode : BOOL;  // if TRUE, the instance afterwards gets moved into the copy code (online change)
END_VAR
AddInput('in0', in0);
AddInput('in1', in1);
AddInput('in2', in2);
AddInput('in3', in3);
AddInput('in4', in4);
AddInput('in5', in5);
AddInput('in6', in6);
AddInput('in7', in7);
AddInput('in8', in8);
AddInput('in9', in9);
AddParameter('index', index);
AddOutput('out',out);
END_METHOD

METHOD PUBLIC  Clone : I_Node
VAR
	pNode : POINTER TO Node_Mux10Way_ITcVnImage;
END_VAR
pNode := __NEW(Node_Mux10Way_ITcVnImage);
Clone := pNode^;
END_METHOD

METHOD PROTECTED OnExecute
CASE index.Value OF
    0: out.TryCopyFrom(in0);
    1: out.TryCopyFrom(in1);
    2: out.TryCopyFrom(in2);
    3: out.TryCopyFrom(in3);
    4: out.TryCopyFrom(in4);
    5: out.TryCopyFrom(in5);
    6: out.TryCopyFrom(in6);
    7: out.TryCopyFrom(in7);
    8: out.TryCopyFrom(in8);
    9: out.TryCopyFrom(in9);
ELSE
    out.Value := 0;
END_CASE
END_METHOD

END_FUNCTION_BLOCK

// Nodes/Image Analysis/Object Detection/Node_F_VN_DetectBlobs
{attribute 'linkalways'} 
{attribute 'no_explicit_call' := 'This FB is a CLASS and must be accessed using methods or properties'}
{attribute 'enable_dynamic_creation'}
FUNCTION_BLOCK Node_F_VN_DetectBlobs EXTENDS VisionNode
VAR
    ipSrcImage : _ITcVnImage;
    ipBlobContours : _ITcVnContainer;
    stParams : _TcVnParamsBlobDetection;
    hrPrev : _HRESULT(S_OK);
	hresult : _HRESULT(S_OK);
END_VAR

METHOD FB_init : BOOL
VAR_INPUT
	bInitRetains : BOOL; // if TRUE, the retain variables are initialized (warm start / cold start)
	bInCopyCode : BOOL;  // if TRUE, the instance afterwards gets moved into the copy code (online change)
END_VAR
AddInput('ipSrcImage', ipSrcImage);
AddInput('stParams', stParams);
AddInput('hrPrev', hrPrev);
AddOutput('ipBlobContours', ipBlobContours);
AddOutput('hresult', hresult);
END_METHOD

METHOD PUBLIC  Clone : I_Node
VAR
	pNode : POINTER TO Node_F_VN_DetectBlobs;
END_VAR
pNode := __NEW(Node_F_VN_DetectBlobs);
Clone := pNode^;
END_METHOD

METHOD PROTECTED OnExecute
hresult.Value := F_VN_DetectBlobs(
	ipSrcImage := ipSrcImage.Value,
    ipBlobContours := ipBlobContours.Value,
    stParams := stParams.Value,
	hrPrev:= hrPrev.Value);
END_METHOD

METHOD PUBLIC PreExecutionCheck
VAR_INPUT
	Check : I_PreExecutionChecks;
END_VAR
Check.IsTrue(ipSrcImage.IsValid, 'ipSrcImage must contain an image');
Check.IsTrue((ipSrcImage.IsPixelDepth(8) OR ipSrcImage.IsPixelDepth(32)), 'ipSrcImage must be 8 or 32 bit pixel depth');
Check.IsTrue((ipSrcImage.HasChannelCount(1) OR ipSrcImage.HasChannelCount(3)), 'ipSrcImage must contain 1 or 3 channels');
Check.IsTrue(stParams.Value.fMaxThreshold >= stParams.Value.fMinThreshold, 'fMaxThreshold must be greater than or equal to fMinThreshold');
END_METHOD

END_FUNCTION_BLOCK

// Nodes/Image Analysis/Object Detection/Node_F_VN_DetectBlobsExp
{attribute 'linkalways'} 
{attribute 'no_explicit_call' := 'This FB is a CLASS and must be accessed using methods or properties'}
{attribute 'enable_dynamic_creation'}
FUNCTION_BLOCK Node_F_VN_DetectBlobsExp EXTENDS VisionNode
VAR
    ipSrcImage : _ITcVnImage;
    ipBlobContours : _ITcVnContainer;
    stParams : _TcVnParamsBlobDetection;
    aOffset : _TcVnPoint;
    hrPrev : _HRESULT(S_OK);
	hresult : _HRESULT(S_OK);
END_VAR

METHOD FB_init : BOOL
VAR_INPUT
	bInitRetains : BOOL; // if TRUE, the retain variables are initialized (warm start / cold start)
	bInCopyCode : BOOL;  // if TRUE, the instance afterwards gets moved into the copy code (online change)
END_VAR
AddInput('ipSrcImage', ipSrcImage);
AddInput('stParams', stParams);
AddInput('aOffset', aOffset);
AddInput('hrPrev', hrPrev);
AddOutput('ipBlobContours', ipBlobContours);
AddOutput('hresult', hresult);
END_METHOD

METHOD PUBLIC  Clone : I_Node
VAR
	pNode : POINTER TO Node_F_VN_DetectBlobsExp;
END_VAR
pNode := __NEW(Node_F_VN_DetectBlobsExp);
Clone := pNode^;
END_METHOD

METHOD PROTECTED OnExecute
hresult.Value := F_VN_DetectBlobsExp(
	ipSrcImage := ipSrcImage.Value,
    ipBlobContours := ipBlobContours.Value,
    stParams := stParams.Value,
    aOffset := aOffset.Value,
	hrPrev:= hrPrev.Value);
END_METHOD

METHOD PUBLIC PreExecutionCheck
VAR_INPUT
	Check : I_PreExecutionChecks;
END_VAR
Check.IsTrue(ipSrcImage.IsValid, 'ipSrcImage must contain an image');
Check.IsTrue((ipSrcImage.IsPixelDepth(8) OR ipSrcImage.IsPixelDepth(32)), 'ipSrcImage must be 8 or 32 bit pixel depth');
Check.IsTrue((ipSrcImage.HasChannelCount(1) OR ipSrcImage.HasChannelCount(3)), 'ipSrcImage must contain 1 or 3 channels');
Check.IsTrue(stParams.Value.fMaxThreshold >= stParams.Value.fMinThreshold, 'fMaxThreshold must be greater than or equal to fMinThreshold');
END_METHOD

END_FUNCTION_BLOCK

// Nodes/Image Analysis/Object Detection/Node_F_VN_FindContourHierarchyExp
{attribute 'linkalways'} 
{attribute 'no_explicit_call' := 'This FB is a CLASS and must be accessed using methods or properties'}
{attribute 'enable_dynamic_creation'}
FUNCTION_BLOCK Node_F_VN_FindContourHierarchyExp EXTENDS VisionNode
VAR
    ipSrcImage : _ITcVnImage;
    ipContours : _ITcVnContainer;
    ipHierarchy : _ITcVnContainer;
    eRetrievalMode : _ETcVnContourRetrievalMode(ETcVnContourRetrievalMode.TCVN_CRM_EXTERNAL);
    eApproximationMethod : _ETcVnContourApproximationMethod(ETcVnContourApproximationMethod.TCVN_CAM_NONE);
    aOffset : _TcVnPoint;
    hrPrev : _HRESULT(S_OK);
	hresult : _HRESULT(S_OK);
END_VAR

METHOD FB_init : BOOL
VAR_INPUT
	bInitRetains : BOOL; // if TRUE, the retain variables are initialized (warm start / cold start)
	bInCopyCode : BOOL;  // if TRUE, the instance afterwards gets moved into the copy code (online change)
END_VAR
AddInput('ipSrcImage', ipSrcImage);
AddParameter('eRetrievalMode', eRetrievalMode);
AddParameter('eApproximationMethod', eApproximationMethod);
AddInput('aOffset', aOffset);
AddInput('hrPrev', hrPrev);
AddOutput('ipContours', ipContours);
AddOutput('ipHierarchy', ipHierarchy);
AddOutput('hresult', hresult);
END_METHOD

METHOD PUBLIC  Clone : I_Node
VAR
	pNode : POINTER TO Node_F_VN_FindContourHierarchyExp;
END_VAR
pNode := __NEW(Node_F_VN_FindContourHierarchyExp);
Clone := pNode^;
END_METHOD

METHOD PROTECTED OnExecute
hresult.Value := F_VN_FindContourHierarchyExp(
	ipSrcImage := ipSrcImage.Value,
    ipContours := ipContours.Value,
    ipHierarchy := ipHierarchy.Value,
    eRetrievalMode := eRetrievalMode.Value,
    eApproximationMethod := eApproximationMethod.Value,
    aOffset := aOffset.Value,
	hrPrev:= hrPrev.Value);
END_METHOD

METHOD PUBLIC PreExecutionCheck
VAR_INPUT
	Check : I_PreExecutionChecks;
END_VAR
Check.IsTrue(ipSrcImage.IsValid, 'ipSrcImage must contain an image');
Check.IsTrue(ipSrcImage.HasChannelCount(1), 'ipSrcImage must contain 1 channel');

IF eRetrievalMode.Value <> ETcVnContourRetrievalMode.TCVN_CRM_FLOODFILL THEN
	RETURN;
END_IF

Check.IsTrue(ipSrcImage.IsElementType(ETcVnElementType.TCVN_ET_DINT), 'ipSrcImage element type must be DINT');
END_METHOD

END_FUNCTION_BLOCK

// Nodes/Image Analysis/Object Detection/Node_F_VN_FindContours
{attribute 'linkalways'} 
{attribute 'no_explicit_call' := 'This FB is a CLASS and must be accessed using methods or properties'}
{attribute 'enable_dynamic_creation'}
FUNCTION_BLOCK Node_F_VN_FindContours EXTENDS VisionNode
VAR
    ipSrcImage : _ITcVnImage;
    ipContours : _ITcVnContainer;
    hrPrev : _HRESULT(S_OK);
	hresult : _HRESULT(S_OK);
END_VAR

METHOD FB_init : BOOL
VAR_INPUT
	bInitRetains : BOOL; // if TRUE, the retain variables are initialized (warm start / cold start)
	bInCopyCode : BOOL;  // if TRUE, the instance afterwards gets moved into the copy code (online change)
END_VAR
AddInput('ipSrcImage', ipSrcImage);
AddInput('hrPrev', hrPrev);
AddOutput('ipContours', ipContours);
AddOutput('hresult', hresult);
END_METHOD

METHOD PUBLIC  Clone : I_Node
VAR
	pNode : POINTER TO Node_F_VN_FindContours;
END_VAR
pNode := __NEW(Node_F_VN_FindContours);
Clone := pNode^;
END_METHOD

METHOD PROTECTED OnExecute
hresult.Value := F_VN_FindContours(
	ipSrcImage := ipSrcImage.Value,
    ipContours := ipContours.Value,
	hrPrev:= hrPrev.Value);
END_METHOD

METHOD PUBLIC PreExecutionCheck
VAR_INPUT
	Check : I_PreExecutionChecks;
END_VAR
Check.IsTrue(ipSrcImage.IsValid, 'ipSrcImage must contain an image');
Check.IsTrue(ipSrcImage.HasChannelCount(1), 'ipSrcImage must contain 1 channel');
END_METHOD

END_FUNCTION_BLOCK

// Nodes/Image Analysis/Object Detection/Node_F_VN_FindContoursExp
{attribute 'linkalways'} 
{attribute 'no_explicit_call' := 'This FB is a CLASS and must be accessed using methods or properties'}
{attribute 'enable_dynamic_creation'}
FUNCTION_BLOCK Node_F_VN_FindContoursExp EXTENDS VisionNode
VAR
    ipSrcImage : _ITcVnImage;
    ipContours : _ITcVnContainer;
    eRetrievalMode : _ETcVnContourRetrievalMode(ETcVnContourRetrievalMode.TCVN_CRM_LIST);
    eApproximationMethod : _ETcVnContourApproximationMethod(ETcVnContourApproximationMethod.TCVN_CAM_NONE);
    aOffset : _TcVnPoint;
    hrPrev : _HRESULT(S_OK);
	hresult : _HRESULT(S_OK);
END_VAR

METHOD FB_init : BOOL
VAR_INPUT
	bInitRetains : BOOL; // if TRUE, the retain variables are initialized (warm start / cold start)
	bInCopyCode : BOOL;  // if TRUE, the instance afterwards gets moved into the copy code (online change)
END_VAR
AddInput('ipSrcImage', ipSrcImage);
AddParameter('eRetrievalMode', eRetrievalMode);
AddParameter('eApproximationMethod', eApproximationMethod);
AddInput('aOffset', aOffset);
AddInput('hrPrev', hrPrev);
AddOutput('ipContours', ipContours);
AddOutput('hresult', hresult);
END_METHOD

METHOD PUBLIC  Clone : I_Node
VAR
	pNode : POINTER TO Node_F_VN_FindContoursExp;
END_VAR
pNode := __NEW(Node_F_VN_FindContoursExp);
Clone := pNode^;
END_METHOD

METHOD PROTECTED OnExecute
hresult.Value := F_VN_FindContoursExp(
	ipSrcImage := ipSrcImage.Value,
    ipContours := ipContours.Value,
    eRetrievalMode := eRetrievalMode.Value,
    eApproximationMethod := eApproximationMethod.Value,
    aOffset := aOffset.Value,
	hrPrev:= hrPrev.Value);
END_METHOD

METHOD PUBLIC PreExecutionCheck
VAR_INPUT
	Check : I_PreExecutionChecks;
END_VAR
Check.IsTrue(ipSrcImage.IsValid, 'ipSrcImage must contain an image');
Check.IsTrue(ipSrcImage.HasChannelCount(1), 'ipSrcImage must contain 1 channel');

IF eRetrievalMode.Value <> ETcVnContourRetrievalMode.TCVN_CRM_FLOODFILL THEN
	RETURN;
END_IF

Check.IsTrue(ipSrcImage.IsElementType(ETcVnElementType.TCVN_ET_DINT), 'ipSrcImage element type must be DINT');
END_METHOD

END_FUNCTION_BLOCK

// Nodes/Image Analysis/Object Detection/Node_F_VN_FindRois
{attribute 'linkalways'}
{attribute 'no_explicit_call' := 'This FB is a CLASS and must be accessed using methods or properties'}
{attribute 'enable_dynamic_creation'}
FUNCTION_BLOCK Node_F_VN_FindRois EXTENDS VisionNode
VAR
    ipSrcImage : _ITcVnImage;
    ipRois : _ITcVnContainer;
    eFindRoisMethod : _ETcVnFindRoisMethod(ETcVnFindRoisMethod.TCVN_FRM_GRID);
    stParams : _TcVnParamsFindRois;
    hrPrev : _HRESULT(S_OK);
    hresult : _HRESULT(S_OK);
END_VAR

METHOD FB_init : BOOL
VAR_INPUT
    bInitRetains : BOOL;
    bInCopyCode : BOOL;
END_VAR
AddInput('ipSrcImage', ipSrcImage);
AddOutput('ipRois', ipRois);
AddParameter('eFindRoisMethod', eFindRoisMethod);
AddInput('stParams', stParams);
AddInput('hrPrev', hrPrev);
AddOutput('hresult', hresult);
END_METHOD

METHOD PUBLIC Clone : I_Node
VAR
    pNode : POINTER TO Node_F_VN_FindRois;
END_VAR
pNode := __NEW(Node_F_VN_FindRois);
Clone := pNode^;
END_METHOD

METHOD PROTECTED OnExecute
hresult.Value := F_VN_FindRois(
    ipSrcImage := ipSrcImage.Value,
    ipRois := ipRois.Value,
    eFindRoisMethod := eFindRoisMethod.Value,
    stParams := stParams.Value,
    hrPrev := hrPrev.Value);
END_METHOD

METHOD PUBLIC PreExecutionCheck
VAR_INPUT
    Check : I_PreExecutionChecks;
END_VAR
Check.IsTrue(ipSrcImage.IsValid, 'ipSrcImage must contain an image');
Check.IsTrue(ipSrcImage.HasChannelCount(1), 'ipSrcImage must contain 1 channel');
Check.IsTrue((eFindRoisMethod.Value = ETcVnFindRoisMethod.TCVN_FRM_GRID) OR
             (eFindRoisMethod.Value = ETcVnFindRoisMethod.TCVN_FRM_CONNECTEDCOMPONENTS), 'Unsupported ROI extraction method');
Check.IsTrue(stParams.Value.stRoiSize.nWidth > 0, 'ROI width must be positive');
Check.IsTrue(stParams.Value.stRoiSize.nHeight > 0, 'ROI height must be positive');
Check.IsTrue((stParams.Value.fMinDensity >= 0.0) AND (stParams.Value.fMinDensity <= 1.0), 'Minimum density must be between 0 and 1');
Check.IsTrue((stParams.Value.fDetectionScaleFactor >= 0.1) AND (stParams.Value.fDetectionScaleFactor <= 1.0), 'Detection scale factor must be between 0.1 and 1');
// Pixel values must be non-negative. Let the API validate pixel content without an additional image scan here.
END_METHOD

END_FUNCTION_BLOCK

// Nodes/Image Analysis/Object Detection/Node_F_VN_FindTemplateWalsh
{attribute 'linkalways'} 
{attribute 'no_explicit_call' := 'This FB is a CLASS and must be accessed using methods or properties'}
{attribute 'enable_dynamic_creation'}
FUNCTION_BLOCK Node_F_VN_FindTemplateWalsh EXTENDS VisionNode
VAR
    ipSrcImage : _ITcVnImage;
    ipTemplateImage : _ITcVnImage;
	ipMatches : _ITcVnContainer;
	fMatchThreshold : _REAL(0.1);
	nProjections : _UDINT(10);
    hrPrev : _HRESULT(S_OK);
	hresult : _HRESULT(S_OK);
END_VAR

METHOD FB_init : BOOL
VAR_INPUT
	bInitRetains : BOOL; // if TRUE, the retain variables are initialized (warm start / cold start)
	bInCopyCode : BOOL;  // if TRUE, the instance afterwards gets moved into the copy code (online change)
END_VAR
AddInput('ipSrcImage', ipSrcImage);
AddInput('ipTemplateImage', ipTemplateImage);
AddInput('fMatchThreshold', fMatchThreshold);
AddInput('nProjections', nProjections);
AddInput('hrPrev', hrPrev);
AddOutput('ipMatches', ipMatches);
AddOutput('hresult',hresult);
END_METHOD

METHOD PUBLIC  Clone : I_Node
VAR
	pNode : POINTER TO Node_F_VN_FindTemplateWalsh;
END_VAR
pNode := __NEW(Node_F_VN_FindTemplateWalsh);
Clone := pNode^;
END_METHOD

METHOD PROTECTED OnExecute
hresult.Value := F_VN_FindTemplateWalsh(
    ipSrcImage := ipSrcImage.Value,
    ipTemplateImage := ipTemplateImage.Value,
	ipMatches := ipMatches.Value,
	fMatchThreshold := fMatchThreshold.Value,
	nProjections := nProjections.Value,
	hrPrev:= hrPrev.Value);
END_METHOD

METHOD PUBLIC PreExecutionCheck
VAR_INPUT
	Check : I_PreExecutionChecks;
END_VAR
Check.IsTrue(ipSrcImage.IsValid, 'ipSrcImage must contain an image');
Check.IsTrue(ipSrcImage.IsPixelDepth(8), 'ipSrcImage must be 8 or 32 bit pixel depth');
Check.IsTrue((ipSrcImage.HasChannelCount(1) OR ipSrcImage.HasChannelCount(3)), 'ipSrcImage must contain 1 or 3 channels');

Check.IsTrue((fMatchThreshold.Value >= 0 AND fMatchThreshold.Value <= 1), 'Threshold must be between 0..1, 1.0 would be a perfect match');

Check.IsTrue(ipTemplateImage.IsValid, 'ipTemplateImage must contain an image');
Check.IsTrue(ImagesHaveMatchingPixelFormats(ipSrcImage.Value, ipTemplateImage.Value), 'ipTemplateImage must have same pixel depth as ipSrcImage');
Check.IsTrue(ImagesHaveMatchingChannels(ipSrcImage.Value, ipTemplateImage.Value), 'ipTemplateImage must have same amount of channels as ipSrcImage');
Check.IsTrue(IsTemplateImageSmallerThanSourceImage(ipSrcImage.Value, ipTemplateImage.Value), 'ipTemplateImage must be smaller than ipSrcImage');
END_METHOD

END_FUNCTION_BLOCK

// Nodes/Image Analysis/Object Detection/Node_F_VN_FindTemplateWalsh_AngleRange
{attribute 'linkalways'} 
{attribute 'no_explicit_call' := 'This FB is a CLASS and must be accessed using methods or properties'}
{attribute 'enable_dynamic_creation'}
FUNCTION_BLOCK Node_F_VN_FindTemplateWalsh_AngleRange EXTENDS VisionNode
VAR
    ipSrcImage : _ITcVnImage;
    ipTemplateImage : _ITcVnImage;
	ipMatches : _ITcVnContainer;
	fMatchThreshold : _REAL(0.1);
	nProjections : _UDINT(10);
	fStartAngle : _LREAL(0);
	fStopAngle : _LREAL(1);
	nAngles : _UDINT(1);
    hrPrev : _HRESULT(S_OK);
	hresult : _HRESULT(S_OK);
END_VAR

METHOD FB_init : BOOL
VAR_INPUT
	bInitRetains : BOOL; // if TRUE, the retain variables are initialized (warm start / cold start)
	bInCopyCode : BOOL;  // if TRUE, the instance afterwards gets moved into the copy code (online change)
END_VAR
AddInput('ipSrcImage', ipSrcImage);
AddInput('ipTemplateImage', ipTemplateImage);
AddInput('fMatchThreshold', fMatchThreshold);
AddInput('nProjections', nProjections);
AddInput('fStartAngle', fStartAngle);
AddInput('fStopAngle', fStopAngle);
AddInput('nAngles', nAngles);
AddInput('hrPrev', hrPrev);
AddOutput('ipMatches', ipMatches);
AddOutput('hresult',hresult);
END_METHOD

METHOD PUBLIC  Clone : I_Node
VAR
	pNode : POINTER TO Node_F_VN_FindTemplateWalsh_AngleRange;
END_VAR
pNode := __NEW(Node_F_VN_FindTemplateWalsh_AngleRange);
Clone := pNode^;
END_METHOD

METHOD PROTECTED OnExecute
hresult.Value := F_VN_FindTemplateWalsh_AngleRange(
    ipSrcImage := ipSrcImage.Value,
    ipTemplateImage := ipTemplateImage.Value,
	ipMatches := ipMatches.Value,
	fMatchThreshold := fMatchThreshold.Value,
	nProjections := nProjections.Value,
	fStartAngle := fStartAngle.Value,
	fStopAngle := fStopAngle.Value,
	nAngles := nAngles.Value,
	hrPrev:= hrPrev.Value);
END_METHOD

METHOD PUBLIC PreExecutionCheck
VAR_INPUT
	Check : I_PreExecutionChecks;
END_VAR
Check.IsTrue(ipSrcImage.IsValid, 'ipSrcImage must contain an image');
Check.IsTrue(ipSrcImage.IsPixelDepth(8), 'ipSrcImage must be 8 or 32 bit pixel depth');
Check.IsTrue((ipSrcImage.HasChannelCount(1) OR ipSrcImage.HasChannelCount(3)), 'ipSrcImage must contain 1 or 3 channels');

Check.IsTrue((fMatchThreshold.Value >= 0 AND fMatchThreshold.Value <= 1), 'Threshold must be between 0..1, 1.0 would be a perfect match');
Check.IsTrue(nProjections.Value <= 50, 'The soft limit of 50 has been reached');

Check.IsTrue(ipTemplateImage.IsValid, 'ipTemplateImage must contain an image');
Check.IsTrue(ImagesHaveMatchingPixelFormats(ipSrcImage.Value, ipTemplateImage.Value), 'ipTemplateImage must have same pixel depth as ipSrcImage');
Check.IsTrue(ImagesHaveMatchingChannels(ipSrcImage.Value, ipTemplateImage.Value), 'ipTemplateImage must have same amount of channels as ipSrcImage');
Check.IsTrue(IsTemplateImageSmallerThanSourceImage(ipSrcImage.Value, ipTemplateImage.Value), 'ipTemplateImage must be smaller than ipSrcImage');
END_METHOD

END_FUNCTION_BLOCK

// Nodes/Image Analysis/Object Detection/Node_F_VN_FindTemplateWalshExp
{attribute 'linkalways'} 
{attribute 'no_explicit_call' := 'This FB is a CLASS and must be accessed using methods or properties'}
{attribute 'enable_dynamic_creation'}
FUNCTION_BLOCK Node_F_VN_FindTemplateWalshExp EXTENDS VisionNode
VAR
    ipSrcImage : _ITcVnImage;
    ipTemplateImage : _ITcVnImage;
	ipMatches : _ITcVnContainer;
	fMatchThreshold : _REAL(0.1);
	nProjections : _UDINT(10);
	eOptions : _ETcVnFindTemplateWalshOptions(ETcVnFindTemplateWalshOptions.TCVN_FTWO_NONE);
	nRotations : _UDINT(1);
	fScaleFactor : _REAL(1);
	eInterpolationType : _ETcVnInterpolationType(ETcVnInterpolationType.TCVN_IT_AREA_BASED);
	ipMatchValues : _ITcVnContainer;
    hrPrev : _HRESULT(S_OK);
	hresult : _HRESULT(S_OK);
END_VAR

